C01815=1200.985,26.673,-44.909,-179.490,5.662,148.847
C01816=1200.990,26.424,-44.893,-179.493,5.662,148.848
C01817=1200.995,26.174,-44.879,-179.495,5.661,148.848
C01818=1201.000,25.924,-44.863,-179.498,5.660,148.849
C01819=1201.005,25.675,-44.848,-179.500,5.660,148.849
C01820=1201.009,25.425,-44.834,-179.503,5.659,148.850
C01821=1201.015,25.176,-44.818,-179.506,5.659,148.851
C01822=1201.019,24.926,-44.803,-179.508,5.658,148.851
C01823=1201.025,24.676,-44.788,-179.510,5.657,148.852
C01824=1201.030,24.427,-44.773,-179.513,5.657,148.853
C01825=1201.035,24.178,-44.758,-179.516,5.656,148.853
C01826=1201.040,23.928,-44.743,-179.518,5.656,148.854
C01827=1201.045,23.679,-44.728,-179.520,5.655,148.854
C01828=1201.050,23.430,-44.713,-179.523,5.654,148.855
C01829=1201.055,23.180,-44.698,-179.526,5.654,148.856
C01830=1201.060,22.931,-44.683,-179.528,5.653,148.856
C01831=1201.065,22.681,-44.669,-179.531,5.653,148.857
C01832=1201.070,22.432,-44.654,-179.533,5.652,148.858
C01833=1201.076,22.182,-44.639,-179.536,5.651,148.858
C01834=1201.080,21.932,-44.623,-179.539,5.651,148.859
C01835=1201.084,21.683,-44.608,-179.541,5.650,148.860
C01836=1201.090,21.433,-44.593,-179.544,5.650,148.860
C01837=1201.095,21.184,-44.578,-179.545,5.650,148.861
C01838=1201.100,20.934,-44.564,-179.548,5.649,148.861
C01839=1201.105,20.685,-44.549,-179.551,5.649,148.862
C01840=1201.110,20.435,-44.534,-179.553,5.648,148.863
C01841=1201.115,20.186,-44.519,-179.556,5.648,148.863
C01842=1201.120,19.936,-44.504,-179.558,5.647,148.864
C01843=1201.125,19.687,-44.489,-179.561,5.646,148.865
C01844=1201.130,19.437,-44.475,-179.563,5.646,148.865
C01845=1201.135,19.188,-44.460,-179.566,5.645,148.866
C01846=1201.140,18.938,-44.445,-179.569,5.645,148.867
C01847=1201.145,18.689,-44.430,-179.571,5.644,148.867
C01848=1201.150,18.439,-44.416,-179.574,5.644,148.868
C01849=1201.156,18.189,-44.401,-179.576,5.643,148.868
C01850=1201.160,17.940,-44.386,-179.579,5.643,148.869
C01851=1201.165,17.690,-44.372,-179.581,5.642,148.870
C01852=1201.170,17.441,-44.357,-179.584,5.641,148.870
C01853=1201.176,17.191,-44.342,-179.586,5.641,148.871
C01854=1201.180,16.942,-44.327,-179.589,5.640,148.872
C01855=1201.185,16.692,-44.313,-179.592,5.640,148.872
C01856=1201.191,16.443,-44.299,-179.594,5.639,148.873
C01857=1201.196,16.194,-44.283,-179.596,5.638,148.873
C01858=1201.201,15.944,-44.269,-179.599,5.638,148.874
C01859=1201.206,15.695,-44.255,-179.601,5.638,148.875
C01860=1201.211,15.446,-44.240,-179.604,5.638,148.876
C01861=1201.216,15.196,-44.225,-179.606,5.637,148.876
C01862=1201.221,14.946,-44.211,-179.609,5.636,148.877
C01863=1201.226,14.697,-44.196,-179.611,5.636,148.877
C01864=1201.231,14.447,-44.181,-179.614,5.635,148.878
C01865=1201.236,14.197,-44.167,-179.617,5.635,148.879
C01866=1201.240,13.948,-44.152,-179.619,5.634,148.879
C01867=1201.245,13.698,-44.138,-179.622,5.634,148.880
C01868=1201.251,13.448,-44.123,-179.624,5.633,148.881
C01869=1201.256,13.199,-44.109,-179.627,5.632,148.881
C01870=1201.261,12.950,-44.094,-179.629,5.632,148.882
C01871=1201.266,12.701,-44.080,-179.632,5.631,148.883
C01872=1201.271,12.451,-44.065,-179.635,5.631,148.883
C01873=1201.276,12.201,-44.051,-179.637,5.630,148.884
C01874=1201.281,11.952,-44.036,-179.639,5.630,148.884
C01875=1201.287,11.702,-44.021,-179.641,5.630,148.885
C01876=1201.291,11.452,-44.007,-179.644,5.629,148.886
C01877=1201.296,11.203,-43.993,-179.647,5.629,148.886
C01878=1201.301,10.954,-43.978,-179.649,5.628,148.887
C01879=1201.307,10.705,-43.964,-179.652,5.627,148.888
C01880=1201.312,10.455,-43.950,-179.654,5.627,148.888
C01881=1201.317,10.205,-43.935,-179.657,5.626,148.889
C01882=1201.322,9.955,-43.921,-179.660,5.626,148.890
C01883=1201.326,9.706,-43.907,-179.662,5.625,148.890
C01884=1201.331,9.457,-43.892,-179.664,5.624,148.891
C01885=1201.337,9.207,-43.877,-179.667,5.624,148.891
C01886=1201.342,8.958,-43.863,-179.669,5.624,148.892
C01887=1201.347,8.708,-43.849,-179.672,5.624,148.893
C01888=1201.352,8.458,-43.834,-179.674,5.623,148.894
C01889=1201.357,8.208,-43.820,-179.677,5.623,148.894
C01890=1201.362,7.959,-43.806,-179.679,5.622,148.895
C01891=1201.367,7.709,-43.792,-179.682,5.621,148.895
C01892=1201.373,7.460,-43.778,-179.684,5.621,148.896
C01893=1201.377,7.211,-43.763,-179.687,5.620,148.897
C01894=1201.382,6.961,-43.748,-179.690,5.620,148.897
C01895=1201.387,6.712,-43.734,-179.692,5.619,148.898
C01896=1201.392,6.462,-43.720,-179.694,5.619,148.899
C01897=1201.397,6.212,-43.706,-179.697,5.619,148.899
C01898=1201.403,5.963,-43.692,-179.699,5.618,148.900
C01899=1201.408,5.713,-43.677,-179.702,5.618,148.901
C01900=1201.413,5.464,-43.663,-179.705,5.617,148.901
C01901=1201.418,5.214,-43.649,-179.707,5.616,148.902
C01902=1201.423,4.964,-43.634,-179.709,5.616,148.902
C01903=1201.428,4.715,-43.621,-179.712,5.615,148.903
C01904=1201.433,4.466,-43.606,-179.715,5.615,148.904
C01905=1201.438,4.216,-43.592,-179.717,5.614,148.905
C01906=1201.442,3.966,-43.578,-179.719,5.615,148.905
C01907=1201.448,3.717,-43.564,-179.722,5.614,148.906
C01908=1201.453,3.468,-43.550,-179.724,5.613,148.906
C01909=1201.458,3.198,-43.535,-179.727,5.613,148.907
C01910=1201.464,2.929,-43.520,-179.730,5.612,148.908
C01911=1201.469,2.660,-43.504,-179.732,5.612,148.908
C01912=1201.475,2.391,-43.490,-179.735,5.611,148.909
C01913=1201.480,2.142,-43.476,-179.738,5.611,148.910
C01914=1201.485,1.892,-43.461,-179.740,5.610,148.910
C01915=1201.490,1.642,-43.447,-179.743,5.610,148.911
C01916=1201.495,1.393,-43.433,-179.746,5.609,148.912
C01917=1201.500,1.144,-43.419,-179.748,5.609,148.913
C01918=1201.505,0.893,-43.405,-179.750,5.608,148.913
C01919=1201.510,0.643,-43.391,-179.752,5.608,148.914
C01920=1201.516,0.394,-43.377,-179.755,5.608,148.914
C01921=1201.520,0.145,-43.363,-179.758,5.607,148.915
C01922=1201.525,-0.105,-43.349,-179.760,5.607,148.916
C01923=1201.531,-0.354,-43.335,-179.763,5.606,148.916
C01924=1201.536,-0.603,-43.321,-179.765,5.605,148.917
C01925=1201.541,-0.854,-43.307,-179.768,5.605,148.918
C01926=1201.546,-1.103,-43.293,-179.770,5.605,148.918
C01927=1201.551,-1.352,-43.280,-179.773,5.605,148.919
C01928=1201.556,-1.602,-43.265,-179.775,5.604,148.920
C01929=1201.561,-1.852,-43.251,-179.778,5.604,148.920
C01930=1201.566,-2.101,-43.238,-179.780,5.603,148.921
C01931=1201.571,-2.351,-43.224,-179.783,5.602,148.921
C01932=1201.576,-2.600,-43.210,-179.785,5.602,148.922
C01933=1201.581,-2.849,-43.196,-179.788,5.602,148.923
C01934=1201.586,-3.100,-43.183,-179.790,5.602,148.924
C01935=1201.591,-3.349,-43.168,-179.793,5.601,148.924
C01936=1201.597,-3.598,-43.154,-179.795,5.600,148.925
C01937=1201.601,-3.848,-43.141,-179.798,5.600,148.925
C01938=1201.606,-4.098,-43.127,-179.800,5.599,148.926
C01939=1201.612,-4.347,-43.113,-179.803,5.599,148.927
C01940=1201.617,-4.597,-43.099,-179.805,5.599,148.927
C01941=1201.622,-4.846,-43.086,-179.808,5.599,148.928
C01942=1201.627,-5.096,-43.072,-179.810,5.598,148.929
C01943=1201.632,-5.345,-43.058,-179.812,5.597,148.929
C01944=1201.638,-5.595,-43.045,-179.815,5.597,148.930
C01945=1201.642,-5.845,-43.031,-179.818,5.596,148.931
C01946=1201.647,-6.094,-43.017,-179.820,5.596,148.931
C01947=1201.653,-6.344,-43.003,-179.822,5.596,148.932
C01948=1201.657,-6.593,-42.990,-179.825,5.596,148.933
C01949=1201.663,-6.842,-42.976,-179.827,5.595,148.933
C01950=1201.668,-7.093,-42.962,-179.830,5.594,148.934
C01951=1201.672,-7.342,-42.949,-179.833,5.594,148.935
C01952=1201.678,-7.592,-42.935,-179.835,5.594,148.935
C01953=1201.683,-7.841,-42.921,-179.837,5.594,148.936
C01954=1201.688,-8.090,-42.908,-179.840,5.593,148.937
C01955=1201.693,-8.340,-42.894,-179.842,5.592,148.937
C01956=1201.698,-8.590,-42.880,-179.845,5.592,148.938
C01957=1201.703,-8.839,-42.867,-179.847,5.592,148.939
C01958=1201.708,-9.089,-42.853,-179.850,5.591,148.939
C01959=1201.714,-9.339,-42.840,-179.852,5.591,148.940
C01960=1201.718,-9.588,-42.826,-179.855,5.591,148.941
C01961=1201.724,-9.837,-42.812,-179.857,5.590,148.941
C01962=1201.729,-10.087,-42.799,-179.860,5.590,148.942
C01963=1201.733,-10.337,-42.785,-179.862,5.589,148.942
C01964=1201.739,-10.586,-42.772,-179.865,5.589,148.943
C01965=1201.743,-10.836,-42.758,-179.867,5.589,148.944
C01966=1201.749,-11.086,-42.745,-179.870,5.588,148.945
C01967=1201.754,-11.335,-42.731,-179.872,5.588,148.945
C01968=1201.759,-11.585,-42.718,-179.875,5.587,148.946
C01969=1201.764,-11.834,-42.704,-179.877,5.587,148.946
C01970=1201.769,-12.084,-42.691,-179.879,5.587,148.947
C01971=1201.774,-12.334,-42.678,-179.882,5.586,148.948
C01972=1201.779,-12.583,-42.664,-179.885,5.586,148.948
C01973=1201.785,-12.833,-42.651,-179.887,5.585,148.949
C01974=1201.790,-13.082,-42.637,-179.890,5.585,148.950
C01975=1201.795,-13.332,-42.624,-179.891,5.585,148.950
C01976=1201.800,-13.582,-42.610,-179.894,5.584,148.951
C01977=1201.805,-13.831,-42.597,-179.897,5.584,148.952
C01978=1201.810,-14.081,-42.583,-179.899,5.583,148.952
C01979=1201.815,-14.330,-42.570,-179.902,5.583,148.953
C01980=1201.820,-14.580,-42.557,-179.905,5.582,148.954
C01981=1201.825,-14.829,-42.543,-179.906,5.582,148.954
C01982=1201.831,-15.079,-42.530,-179.909,5.582,148.955
C01983=1201.835,-15.329,-42.517,-179.912,5.581,148.956
C01984=1201.841,-15.578,-42.503,-179.914,5.581,148.956
C01985=1201.845,-15.828,-42.490,-179.917,5.581,148.957
C01986=1201.851,-16.077,-42.477,-179.919,5.581,148.958
C01987=1201.855,-16.327,-42.463,-179.922,5.580,148.958
C01988=1201.861,-16.576,-42.450,-179.924,5.580,148.959
C01989=1201.866,-16.826,-42.437,-179.927,5.579,148.960
C01990=1201.871,-17.075,-42.423,-179.929,5.579,148.960
C01991=1201.876,-17.325,-42.410,-179.931,5.579,148.961
C01992=1201.882,-17.575,-42.397,-179.934,5.578,148.962
C01993=1201.886,-17.825,-42.384,-179.937,5.578,148.962
C01994=1201.892,-18.074,-42.370,-179.939,5.577,148.963
C01995=1201.897,-18.323,-42.358,-179.941,5.577,148.963
C01996=1201.902,-18.574,-42.344,-179.943,5.577,148.964
C01997=1201.907,-18.823,-42.331,-179.946,5.576,148.965
C01998=1201.912,-19.072,-42.318,-179.949,5.576,148.966
C01999=1201.917,-19.322,-42.305,-179.951,5.575,148.966
C02000=1201.922,-19.572,-42.292,-179.954,5.576,148.967
C02001=1201.928,-19.822,-42.278,-179.956,5.575,148.967
C02002=1201.933,-20.070,-42.265,-179.958,5.574,148.968
C02003=1201.937,-20.320,-42.252,-179.961,5.574,148.969
C02004=1201.943,-20.570,-42.239,-179.964,5.574,148.970
C02005=1201.947,-20.820,-42.226,-179.966,5.574,148.970
C02006=1201.953,-21.070,-42.213,-179.968,5.573,148.971
C02007=1201.958,-21.318,-42.200,-179.971,5.573,148.972
C02008=1201.963,-21.568,-42.187,-179.973,5.572,148.972
C02009=1201.969,-21.818,-42.173,-179.975,5.572,148.973
C02010=1201.973,-22.068,-42.160,-179.978,5.572,148.973
C02011=1201.978,-22.317,-42.148,-179.981,5.571,148.974
C02012=1201.984,-22.567,-42.135,-179.983,5.571,148.975
C02013=1201.989,-22.836,-42.120,-179.986,5.570,148.976
C02014=1201.994,-23.106,-42.106,-179.989,5.570,148.976
C02015=1202.000,-23.375,-42.093,-179.991,5.570,148.977
C02016=1202.006,-23.645,-42.078,-179.993,5.570,148.978
C02017=1202.011,-23.895,-42.066,-179.996,5.569,148.978
C02018=1202.016,-24.145,-42.052,-179.999,5.569,148.979
C02019=1202.021,-24.394,-42.040,179.999,5.568,148.980
C02020=1202.026,-24.644,-42.026,179.997,5.569,148.980
C02021=1202.031,-24.893,-42.013,179.994,5.568,148.981
C02022=1202.037,-25.143,-42.000,179.992,5.567,148.982
C02023=1202.041,-25.393,-41.987,179.989,5.567,148.982
C02024=1202.046,-25.642,-41.975,179.986,5.567,148.983
C02025=1202.052,-25.892,-41.961,179.984,5.567,148.984
C02026=1202.057,-26.142,-41.948,179.982,5.566,148.984
C02027=1202.062,-26.391,-41.936,179.979,5.566,148.985
C02028=1202.067,-26.640,-41.923,179.977,5.565,148.986
C02029=1202.072,-26.891,-41.910,179.975,5.565,148.986
C02030=1202.077,-27.140,-41.897,179.972,5.565,148.987
C02031=1202.082,-27.389,-41.884,179.969,5.564,148.988
C02032=1202.087,-27.638,-41.872,179.967,5.564,148.988
C02033=1202.093,-27.889,-41.858,179.965,5.564,148.989
C02034=1202.098,-28.138,-41.846,179.963,5.563,148.989
C02035=1202.103,-28.387,-41.833,179.960,5.563,148.990
C02036=1202.107,-28.637,-41.820,179.957,5.563,148.991
C02037=1202.113,-28.887,-41.807,179.955,5.563,148.992
C02038=1202.118,-29.136,-41.794,179.952,5.562,148.992
C02039=1202.124,-29.386,-41.782,179.950,5.562,148.993
C02040=1202.128,-29.636,-41.769,179.947,5.561,148.994
C02041=1202.134,-29.886,-41.757,179.946,5.561,148.994
C02042=1202.139,-30.135,-41.744,179.943,5.561,148.995
C02043=1202.144,-30.385,-41.731,179.940,5.560,148.996
C02044=1202.149,-30.635,-41.718,179.938,5.560,148.996
C02045=1202.154,-30.884,-41.705,179.935,5.560,148.997
C02046=1202.159,-31.133,-41.693,179.933,5.560,148.998
C02047=1202.164,-31.383,-41.680,179.930,5.559,148.998
C02048=1202.169,-31.633,-41.667,179.929,5.559,148.999
C02049=1202.175,-31.883,-41.655,179.926,5.559,148.999
C02050=1202.180,-32.132,-41.642,179.923,5.558,149.000
C02051=1202.185,-32.382,-41.629,179.921,5.558,149.001
C02052=1202.190,-32.631,-41.617,179.919,5.558,149.002
C02053=1202.195,-32.881,-41.604,179.916,5.558,149.002
C02054=1202.200,-33.131,-41.592,179.913,5.557,149.003
C02055=1202.206,-33.380,-41.580,179.911,5.557,149.003
C02056=1202.211,-33.630,-41.566,179.909,5.557,149.004
C02057=1202.216,-33.880,-41.553,179.906,5.556,149.005
C02058=1202.221,-34.129,-41.541,179.904,5.556,149.006
C02059=1202.227,-34.379,-41.529,179.902,5.556,149.006
C02060=1202.232,-34.628,-41.516,179.899,5.556,149.007
C02061=1202.236,-34.878,-41.503,179.896,5.555,149.008
C02062=1202.241,-35.128,-41.491,179.894,5.555,149.008
C02063=1202.247,-35.378,-41.479,179.892,5.555,149.009
C02064=1202.252,-35.627,-41.466,179.889,5.554,149.010
C02065=1202.257,-35.876,-41.454,179.887,5.554,149.010
C02066=1202.261,-36.126,-41.441,179.884,5.553,149.011
C02067=1202.267,-36.376,-41.429,179.882,5.554,149.012
C02068=1202.272,-36.625,-41.416,179.880,5.553,149.012
C02069=1202.278,-36.875,-41.403,179.877,5.552,149.013
C02070=1202.283,-37.125,-41.391,179.875,5.553,149.013
C02071=1202.288,-37.374,-41.378,179.872,5.552,149.014
C02072=1202.293,-37.624,-41.366,179.870,5.552,149.015
C02073=1202.298,-37.874,-41.353,179.867,5.551,149.016
C02074=1202.304,-38.124,-41.341,179.865,5.552,149.016
C02075=1202.309,-38.373,-41.328,179.863,5.551,149.017
C02076=1202.314,-38.623,-41.317,179.860,5.550,149.017
C02077=1202.319,-38.872,-41.304,179.858,5.551,149.018
C02078=1202.324,-39.121,-41.291,179.855,5.550,149.019
C02079=1202.329,-39.372,-41.279,179.853,5.550,149.020
C02080=1202.334,-39.621,-41.267,179.850,5.549,149.020
C02081=1202.339,-39.871,-41.254,179.848,5.550,149.021
C02082=1202.345,-40.121,-41.242,179.846,5.549,149.021
C02083=1202.350,-40.370,-41.229,179.843,5.548,149.022
C02084=1202.355,-40.620,-41.218,179.841,5.549,149.023
C02085=1202.360,-40.869,-41.206,179.838,5.548,149.024
C02086=1202.365,-41.118,-41.193,179.836,5.548,149.024
C02087=1202.370,-41.369,-41.181,179.834,5.548,149.025
C02088=1202.375,-41.618,-41.168,179.831,5.547,149.025
C02089=1202.380,-41.868,-41.156,179.829,5.547,149.026
C02090=1202.385,-42.117,-41.144,179.826,5.547,149.027
C02091=1202.391,-42.367,-41.132,179.824,5.547,149.028
C02092=1202.396,-42.617,-41.119,179.821,5.546,149.028
C02093=1202.401,-42.867,-41.107,179.819,5.546,149.029
C02094=1202.407,-43.116,-41.095,179.817,5.546,149.030
C02095=1202.412,-43.366,-41.083,179.814,5.545,149.030
C02096=1202.417,-43.615,-41.070,179.812,5.545,149.031
C02097=1202.422,-43.865,-41.059,179.810,5.545,149.031
C02098=1202.426,-44.115,-41.046,179.807,5.545,149.032
C02099=1202.432,-44.365,-41.034,179.804,5.544,149.033
C02100=1202.437,-44.614,-41.021,179.802,5.545,149.034
C02101=1202.442,-44.864,-41.010,179.800,5.544,149.034
C02102=1202.447,-45.113,-40.997,179.797,5.543,149.035
C02103=1202.453,-45.363,-40.985,179.795,5.543,149.035
C02104=1202.458,-45.613,-40.972,179.793,5.543,149.036
C02105=1202.463,-45.862,-40.961,179.790,5.543,149.037
C02106=1202.468,-46.112,-40.949,179.787,5.542,149.038
C02107=1202.473,-46.362,-40.937,179.785,5.543,149.038
C02108=1202.479,-46.611,-40.925,179.783,5.542,149.039
C02109=1202.484,-46.861,-40.912,179.780,5.542,149.039
C02110=1202.489,-47.111,-40.900,179.778,5.542,149.040
C02111=1202.494,-47.360,-40.889,179.776,5.541,149.041
C02112=1202.499,-47.610,-40.876,179.773,5.541,149.042
C02113=1202.504,-47.860,-40.864,179.771,5.541,149.042
C02114=1202.510,-48.109,-40.852,179.769,5.540,149.043
C02115=1202.515,-48.359,-40.840,179.766,5.540,149.043
C02116=1202.520,-48.608,-40.829,179.764,5.540,149.044
C02117=1202.526,-48.879,-40.815,179.761,5.540,149.045
C02118=1202.532,-49.149,-40.803,179.759,5.539,149.046
C02119=1202.537,-49.419,-40.789,179.756,5.539,149.046
C02120=1202.542,-49.689,-40.776,179.753,5.539,149.047
C02121=1202.547,-49.939,-40.764,179.751,5.539,149.048
C02122=1202.552,-50.188,-40.753,179.749,5.538,149.048
C02123=1202.557,-50.438,-40.740,179.746,5.538,149.049
C02124=1202.563,-50.688,-40.728,179.744,5.538,149.050
C02125=1202.568,-50.938,-40.716,179.741,5.538,149.050
C02126=1202.573,-51.187,-40.705,179.739,5.537,149.051
C02127=1202.578,-51.437,-40.692,179.737,5.537,149.052
C02128=1202.584,-51.686,-40.681,179.734,5.537,149.052
C02129=1202.589,-51.936,-40.669,179.732,5.537,149.053
C02130=1202.594,-52.185,-40.658,179.730,5.537,149.054
C02131=1202.599,-52.435,-40.645,179.727,5.536,149.054
C02132=1202.605,-52.685,-40.633,179.724,5.536,149.055
C02133=1202.609,-52.934,-40.622,179.723,5.536,149.056
C02134=1202.615,-53.184,-40.610,179.720,5.535,149.056
C02135=1202.620,-53.434,-40.598,179.717,5.535,149.057
C02136=1202.624,-53.683,-40.586,179.715,5.535,149.058
C02137=1202.630,-53.933,-40.574,179.712,5.535,149.058
C02138=1202.635,-54.183,-40.562,179.710,5.535,149.059
C02139=1202.640,-54.433,-40.551,179.708,5.534,149.060
C02140=1202.645,-54.682,-40.539,179.706,5.534,149.060
C02141=1202.651,-54.932,-40.527,179.703,5.534,149.061
C02142=1202.655,-55.182,-40.515,179.701,5.534,149.062
C02143=1202.661,-55.431,-40.504,179.698,5.533,149.062
C02144=1202.666,-55.681,-40.492,179.696,5.534,149.063
C02145=1202.671,-55.930,-40.481,179.694,5.533,149.064
C02146=1202.677,-56.180,-40.469,179.691,5.533,149.064
C02147=1202.682,-56.430,-40.456,179.689,5.533,149.065
C02148=1202.687,-56.679,-40.445,179.686,5.532,149.066
C02149=1202.692,-56.929,-40.433,179.684,5.532,149.066
C02150=1202.697,-57.179,-40.422,179.682,5.532,149.067
C02151=1202.702,-57.429,-40.410,179.680,5.532,149.068
C02152=1202.708,-57.679,-40.398,179.677,5.531,149.068
C02153=1202.712,-57.928,-40.387,179.675,5.531,149.069
C02154=1202.718,-58.178,-40.375,179.672,5.531,149.070
C02155=1202.723,-58.427,-40.364,179.670,5.531,149.070
C02156=1202.728,-58.677,-40.352,179.667,5.531,149.071
C02157=1202.733,-58.927,-40.341,179.665,5.530,149.072
C02158=1202.738,-59.176,-40.328,179.663,5.530,149.072
C02159=1202.744,-59.426,-40.316,179.660,5.530,149.073
C02160=1202.748,-59.676,-40.305,179.658,5.530,149.074
C02161=1202.754,-59.925,-40.293,179.656,5.530,149.074
C02162=1202.759,-60.174,-40.282,179.653,5.529,149.075
C02163=1202.765,-60.424,-40.270,179.651,5.529,149.076
C02164=1202.769,-60.674,-40.259,179.649,5.529,149.076
C02165=1202.775,-60.924,-40.247,179.646,5.529,149.077
C02166=1202.779,-61.174,-40.236,179.644,5.529,149.078
C02167=1202.785,-61.423,-40.224,179.641,5.528,149.078
C02168=1202.790,-61.672,-40.213,179.639,5.528,149.079
C02169=1202.796,-61.922,-40.201,179.637,5.528,149.080
C02170=1202.801,-62.173,-40.190,179.634,5.528,149.080
C02171=1202.806,-62.423,-40.179,179.632,5.527,149.081
C02172=1202.811,-62.672,-40.167,179.630,5.527,149.082
C02173=1202.817,-62.921,-40.156,179.627,5.527,149.082
C02174=1202.821,-63.171,-40.145,179.625,5.527,149.083
C02175=1202.827,-63.421,-40.133,179.623,5.527,149.084
C02176=1202.832,-63.671,-40.121,179.620,5.526,149.084
C02177=1202.837,-63.921,-40.109,179.618,5.526,149.085
C02178=1202.842,-64.169,-40.099,179.615,5.526,149.086
C02179=1202.848,-64.419,-40.087,179.613,5.526,149.086
C02180=1202.852,-64.669,-40.075,179.611,5.526,149.087
C02181=1202.858,-64.919,-40.063,179.608,5.525,149.088
C02182=1202.863,-65.169,-40.053,179.606,5.526,149.088
C02183=1202.869,-65.418,-40.041,179.604,5.525,149.089
C02184=1202.874,-65.668,-40.030,179.601,5.525,149.090
C02185=1202.878,-65.918,-40.019,179.599,5.525,149.090
C02186=1202.884,-66.168,-40.007,179.597,5.524,149.091
C02187=1202.889,-66.417,-39.996,179.594,5.524,149.092
C02188=1202.894,-66.666,-39.984,179.592,5.524,149.092
C02189=1202.899,-66.917,-39.974,179.589,5.524,149.093
C02190=1202.904,-67.166,-39.962,179.587,5.524,149.094
C02191=1202.910,-67.416,-39.951,179.585,5.524,149.094
C02192=1202.915,-67.665,-39.939,179.582,5.523,149.095
C02193=1202.920,-67.915,-39.928,179.580,5.523,149.096
C02194=1202.925,-68.165,-39.917,179.578,5.523,149.096
C02195=1202.930,-68.414,-39.906,179.576,5.523,149.097
C02196=1202.936,-68.664,-39.894,179.573,5.523,149.098
C02197=1202.941,-68.914,-39.883,179.571,5.522,149.098
C02198=1202.947,-69.164,-39.872,179.569,5.522,149.099
C02199=1202.952,-69.413,-39.861,179.566,5.522,149.100
C02200=1202.956,-69.663,-39.849,179.564,5.522,149.100
C02201=1202.962,-69.913,-39.838,179.561,5.522,149.101
C02202=1202.967,-70.162,-39.827,179.559,5.521,149.102
C02203=1202.972,-70.412,-39.816,179.557,5.521,149.102
C02204=1202.977,-70.662,-39.804,179.554,5.521,149.103
C02205=1202.983,-70.911,-39.793,179.552,5.521,149.104
C02206=1202.988,-71.161,-39.783,179.549,5.521,149.104
C02207=1202.993,-71.411,-39.771,179.547,5.520,149.105
C02208=1202.998,-71.660,-39.760,179.545,5.520,149.106
C02209=1203.003,-71.910,-39.749,179.543,5.520,149.106
C02210=1203.009,-72.160,-39.737,179.540,5.520,149.107
C02211=1203.014,-72.409,-39.727,179.538,5.520,149.108
C02212=1203.019,-72.659,-39.716,179.535,5.519,149.108
C02213=1203.024,-72.909,-39.705,179.533,5.519,149.109
C02214=1203.030,-73.158,-39.693,179.531,5.519,149.110
C02215=1203.035,-73.409,-39.683,179.529,5.519,149.110
C02216=1203.040,-73.658,-39.671,179.526,5.519,149.111
C02217=1203.046,-73.908,-39.660,179.523,5.518,149.112
C02218=1203.051,-74.158,-39.649,179.522,5.518,149.112
C02219=1203.055,-74.407,-39.638,179.519,5.518,149.113
C02220=1203.061,-74.657,-39.628,179.517,5.518,149.114
C02221=1203.067,-74.928,-39.615,179.514,5.518,149.114
C02222=1203.072,-75.199,-39.603,179.512,5.517,149.115
C02223=1203.078,-75.469,-39.591,179.510,5.518,149.116
C02224=1203.083,-75.740,-39.580,179.507,5.517,149.116
C02225=1203.089,-75.990,-39.568,179.504,5.517,149.117
C02226=1203.094,-76.239,-39.558,179.502,5.517,149.118
C02227=1203.099,-76.489,-39.546,179.500,5.517,149.119
C02228=1203.105,-76.738,-39.536,179.497,5.516,149.119
C02229=1203.110,-76.988,-39.524,179.495,5.516,149.120
C02230=1203.115,-77.239,-39.514,179.493,5.516,149.120
C02231=1203.120,-77.487,-39.503,179.490,5.516,149.121
C02232=1203.125,-77.738,-39.492,179.488,5.516,149.122
C02233=1203.131,-77.987,-39.481,179.486,5.516,149.122
C02234=1203.136,-78.237,-39.470,179.484,5.515,149.123
C02235=1203.141,-78.487,-39.459,179.481,5.515,149.124
C02236=1203.147,-78.736,-39.448,179.479,5.515,149.124
C02237=1203.151,-78.986,-39.437,179.476,5.515,149.125
C02238=1203.157,-79.236,-39.427,179.475,5.515,149.126
C02239=1203.162,-79.485,-39.416,179.472,5.515,149.126
C02240=1203.168,-79.735,-39.405,179.470,5.515,149.127
C02241=1203.173,-79.985,-39.394,179.467,5.514,149.128
C02242=1203.178,-80.235,-39.383,179.465,5.514,149.128
C02243=1203.183,-80.484,-39.372,179.463,5.514,149.129
C02244=1203.188,-80.734,-39.362,179.460,5.514,149.130
C02245=1203.194,-80.984,-39.351,179.458,5.514,149.130
C02246=1203.198,-81.233,-39.340,179.455,5.514,149.131
C02247=1203.204,-81.483,-39.330,179.454,5.514,149.132
C02248=1203.209,-81.733,-39.318,179.451,5.513,149.132
C02249=1203.214,-81.983,-39.307,179.448,5.513,149.133
C02250=1203.220,-82.232,-39.297,179.446,5.513,149.134
C02251=1203.225,-82.482,-39.286,179.444,5.513,149.134
C02252=1203.230,-82.732,-39.276,179.442,5.513,149.135
C02253=1203.235,-82.981,-39.264,179.439,5.512,149.136
C02254=1203.240,-83.231,-39.254,179.437,5.513,149.136
C02255=1203.245,-83.481,-39.244,179.435,5.512,149.137
C02256=1203.251,-83.730,-39.233,179.432,5.512,149.138
C02257=1203.256,-83.980,-39.222,179.430,5.512,149.138
C02258=1203.261,-84.230,-39.212,179.428,5.511,149.139
C02259=1203.266,-84.479,-39.201,179.426,5.512,149.140
C02260=1203.272,-84.729,-39.190,179.423,5.511,149.140
C02261=1203.277,-84.979,-39.180,179.421,5.511,149.141
C02262=1203.283,-85.228,-39.168,179.419,5.511,149.142
C02263=1203.288,-85.479,-39.158,179.417,5.511,149.142
C02264=1203.293,-85.728,-39.148,179.414,5.511,149.143
C02265=1203.298,-85.978,-39.137,179.411,5.510,149.144
C02266=1203.303,-86.227,-39.126,179.410,5.510,149.144
C02267=1203.308,-86.478,-39.115,179.407,5.510,149.145
C02268=1203.314,-86.727,-39.105,179.405,5.510,149.146
C02269=1203.319,-86.977,-39.094,179.402,5.510,149.146
C02270=1203.324,-87.226,-39.084,179.401,5.510,149.147
C02271=1203.329,-87.477,-39.073,179.398,5.509,149.148
C02272=1203.335,-87.726,-39.063,179.396,5.510,149.148
C02273=1203.340,-87.976,-39.052,179.393,5.509,149.149
C02274=1203.345,-88.225,-39.041,179.391,5.509,149.149
C02275=1203.350,-88.476,-39.031,179.389,5.509,149.150
C02276=1203.356,-88.725,-39.021,179.386,5.508,149.151
C02277=1203.360,-88.975,-39.011,179.384,5.509,149.152
C02278=1203.365,-89.224,-39.000,179.381,5.508,149.152
C02279=1203.371,-89.473,-38.990,179.380,5.508,149.153
C02280=1203.376,-89.724,-38.979,179.377,5.508,149.153
C02281=1203.382,-89.973,-38.969,179.375,5.508,149.154
C02282=1203.387,-90.224,-38.958,179.372,5.508,149.155
C02283=1203.392,-90.472,-38.947,179.371,5.508,149.155
C02284=1203.397,-90.723,-38.937,179.368,5.508,149.156
C02285=1203.402,-90.972,-38.926,179.366,5.507,149.157
C02286=1203.407,-91.222,-38.916,179.363,5.507,149.157
C02287=1203.413,-91.472,-38.906,179.361,5.507,149.158
C02288=1203.419,-91.722,-38.895,179.359,5.507,149.159
C02289=1203.424,-91.972,-38.885,179.356,5.507,149.159
C02290=1203.429,-92.221,-38.875,179.354,5.507,149.160
C02291=1203.433,-92.471,-38.864,179.352,5.506,149.161
C02292=1203.439,-92.720,-38.854,179.350,5.507,149.161
C02293=1203.444,-92.970,-38.844,179.347,5.506,149.162
C02294=1203.449,-93.220,-38.833,179.345,5.507,149.163
C02295=1203.455,-93.470,-38.823,179.343,5.506,149.163
C02296=1203.460,-93.720,-38.812,179.341,5.506,149.164
C02297=1203.466,-93.969,-38.802,179.338,5.506,149.165
C02298=1203.471,-94.219,-38.792,179.336,5.506,149.165
C02299=1203.476,-94.469,-38.781,179.334,5.505,149.166
C02300=1203.481,-94.718,-38.772,179.331,5.505,149.167
C02301=1203.487,-94.968,-38.761,179.329,5.505,149.167
C02302=1203.492,-95.218,-38.751,179.327,5.505,149.168
C02303=1203.497,-95.468,-38.741,179.325,5.505,149.168
C02304=1203.502,-95.718,-38.730,179.322,5.504,149.169
C02305=1203.508,-95.967,-38.720,179.320,5.505,149.170
C02306=1203.513,-96.217,-38.710,179.318,5.504,149.171
C02307=1203.518,-96.467,-38.700,179.316,5.504,149.171
C02308=1203.523,-96.716,-38.689,179.313,5.504,149.172
C02309=1203.529,-96.966,-38.679,179.311,5.504,149.172
C02310=1203.534,-97.216,-38.669,179.309,5.504,149.173
C02311=1203.539,-97.465,-38.659,179.307,5.504,149.174
C02312=1203.544,-97.715,-38.649,179.304,5.504,149.174
C02313=1203.549,-97.965,-38.638,179.302,5.504,149.175
C02314=1203.555,-98.215,-38.628,179.300,5.503,149.176
C02315=1203.561,-98.464,-38.618,179.298,5.503,149.176
C02316=1203.565,-98.714,-38.608,179.295,5.503,149.177
C02317=1203.570,-98.964,-38.598,179.293,5.503,149.178
C02318=1203.576,-99.213,-38.587,179.291,5.503,149.178
C02319=1203.581,-99.464,-38.577,179.288,5.502,149.179
C02320=1203.586,-99.713,-38.567,179.286,5.503,149.180
C02321=1203.591,-99.962,-38.557,179.284,5.502,149.180
C02322=1203.596,-100.213,-38.546,179.282,5.503,149.181
C02323=1203.602,-100.463,-38.537,179.279,5.502,149.182
C02324=1203.607,-100.712,-38.527,179.277,5.502,149.182
C02325=1203.613,-100.984,-38.516,179.275,5.502,149.183
C02326=1203.618,-101.255,-38.505,179.272,5.502,149.184
C02327=1203.625,-101.526,-38.494,179.270,5.502,149.184
C02328=1203.630,-101.797,-38.483,179.267,5.501,149.185
C02329=1203.636,-102.047,-38.473,179.265,5.502,149.186
C02330=1203.640,-102.297,-38.463,179.263,5.501,149.186
C02331=1203.646,-102.547,-38.453,179.261,5.501,149.187
C02332=1203.651,-102.796,-38.443,179.258,5.501,149.188
C02333=1203.656,-103.046,-38.433,179.256,5.501,149.188
C02334=1203.661,-103.296,-38.423,179.254,5.500,149.189
C02335=1203.667,-103.546,-38.413,179.252,5.501,149.190
C02336=1203.673,-103.796,-38.403,179.249,5.500,149.190
C02337=1203.678,-104.045,-38.393,179.247,5.500,149.191
C02338=1203.683,-104.295,-38.383,179.245,5.500,149.192
C02339=1203.688,-104.544,-38.373,179.243,5.500,149.192
C02340=1203.693,-104.794,-38.364,179.240,5.500,149.193
C02341=1203.699,-105.044,-38.354,179.238,5.500,149.193
C02342=1203.703,-105.294,-38.344,179.236,5.500,149.194
C02343=1203.709,-105.543,-38.333,179.234,5.500,149.195
C02344=1203.715,-105.794,-38.324,179.231,5.499,149.195
C02345=1203.720,-106.043,-38.314,179.229,5.500,149.196
C02346=1203.725,-106.293,-38.304,179.227,5.499,149.197
C02347=1203.730,-106.543,-38.293,179.225,5.500,149.198
C02348=1203.735,-106.792,-38.285,179.222,5.499,149.198
C02349=1203.741,-107.042,-38.274,179.220,5.499,149.199
C02350=1203.745,-107.292,-38.264,179.218,5.499,149.199
C02351=1203.751,-107.542,-38.255,179.216,5.499,149.200
C02352=1203.757,-107.792,-38.245,179.213,5.498,149.201
C02353=1203.762,-108.041,-38.235,179.211,5.499,149.201
C02354=1203.768,-108.291,-38.226,179.209,5.498,149.202
C02355=1203.772,-108.541,-38.216,179.207,5.498,149.203
C02356=1203.777,-108.790,-38.205,179.204,5.498,149.203
C02357=1203.783,-109.040,-38.195,179.202,5.498,149.204
C02358=1203.788,-109.290,-38.186,179.200,5.497,149.204
C02359=1203.794,-109.539,-38.176,179.198,5.498,149.205
C02360=1203.799,-109.789,-38.167,179.195,5.497,149.206
C02361=1203.804,-110.040,-38.157,179.194,5.497,149.206
C02362=1203.809,-110.289,-38.147,179.191,5.497,149.207
C02363=1203.815,-110.539,-38.137,179.189,5.497,149.208
C02364=1203.820,-110.788,-38.128,179.187,5.497,149.208
C02365=1203.825,-111.038,-38.118,179.185,5.497,149.209
C02366=1203.831,-111.288,-38.108,179.182,5.497,149.210
C02367=1203.835,-111.538,-38.098,179.180,5.497,149.210
C02368=1203.841,-111.788,-38.089,179.178,5.496,149.211
C02369=1203.846,-112.037,-38.079,179.176,5.497,149.212
C02370=1203.852,-112.287,-38.069,179.173,5.496,149.212
C02371=1203.857,-112.537,-38.060,179.171,5.496,149.213
C02372=1203.862,-112.786,-38.050,179.169,5.496,149.214
C02373=1203.868,-113.036,-38.041,179.167,5.496,149.214
C02374=1203.873,-113.286,-38.030,179.164,5.495,149.215
C02375=1203.878,-113.536,-38.021,179.162,5.496,149.215
C02376=1203.883,-113.786,-38.011,179.160,5.495,149.216
C02377=1203.889,-114.035,-38.002,179.158,5.495,149.217
C02378=1203.894,-114.285,-37.992,179.155,5.495,149.217
C02379=1203.899,-114.535,-37.983,179.153,5.495,149.218
C02380=1203.905,-114.784,-37.973,179.151,5.495,149.219
C02381=1203.910,-115.034,-37.964,179.149,5.495,149.219
C02382=1203.914,-115.284,-37.954,179.146,5.495,149.220
C02383=1203.920,-115.534,-37.945,179.145,5.495,149.220
C02384=1203.925,-115.784,-37.935,179.142,5.494,149.221
C02385=1203.931,-116.034,-37.925,179.140,5.495,149.222
C02386=1203.936,-116.283,-37.916,179.138,5.494,149.222
C02387=1203.942,-116.533,-37.906,179.136,5.494,149.223
C02388=1203.947,-116.782,-37.897,179.134,5.495,149.224
C02389=1203.953,-117.033,-37.887,179.131,5.494,149.224
C02390=1203.957,-117.282,-37.878,179.129,5.494,149.225
C02391=1203.963,-117.532,-37.869,179.127,5.494,149.226
C02392=1203.968,-117.781,-37.859,179.125,5.494,149.226
C02393=1203.973,-118.032,-37.849,179.122,5.493,149.227
C02394=1203.979,-118.282,-37.840,179.120,5.494,149.228
C02395=1203.983,-118.531,-37.830,179.118,5.493,149.228
C02396=1203.989,-118.781,-37.821,179.116,5.493,149.229
C02397=1203.994,-119.031,-37.811,179.113,5.493,149.230
C02398=1203.999,-119.280,-37.802,179.112,5.493,149.230
C02399=1204.005,-119.530,-37.793,179.109,5.493,149.231
C02400=1204.010,-119.780,-37.783,179.107,5.493,149.232
C02401=1204.015,-120.030,-37.774,179.105,5.492,149.232
C02402=1204.021,-120.279,-37.764,179.103,5.493,149.233
C02403=1204.026,-120.529,-37.755,179.100,5.492,149.233
C02404=1204.031,-120.779,-37.746,179.098,5.492,149.234
C02405=1204.037,-121.028,-37.736,179.096,5.492,149.235
C02406=1204.042,-121.278,-37.727,179.094,5.492,149.235
C02407=1204.047,-121.528,-37.718,179.092,5.492,149.236
C02408=1204.053,-121.778,-37.708,179.089,5.492,149.237
C02409=1204.058,-122.027,-37.699,179.087,5.492,149.237
C02410=1204.063,-122.277,-37.690,179.085,5.491,149.238
C02411=1204.069,-122.527,-37.680,179.083,5.492,149.238
C02412=1204.074,-122.777,-37.671,179.080,5.491,149.239
C02413=1204.079,-123.027,-37.662,179.079,5.491,149.240
C02414=1204.085,-123.277,-37.653,179.076,5.491,149.240
C02415=1204.090,-123.526,-37.643,179.074,5.491,149.241
C02416=1204.095,-123.776,-37.634,179.072,5.491,149.242
C02417=1204.100,-124.026,-37.625,179.070,5.491,149.242
C02418=1204.106,-124.275,-37.615,179.067,5.490,149.243
C02419=1204.111,-124.525,-37.606,179.065,5.491,149.244
C02420=1204.116,-124.775,-37.597,179.063,5.490,149.244
C02421=1204.122,-125.025,-37.588,179.061,5.490,149.245
C02422=1204.127,-125.274,-37.578,179.059,5.491,149.245
C02423=1204.132,-125.524,-37.569,179.056,5.490,149.246
C02424=1204.137,-125.774,-37.560,179.055,5.490,149.247
C02425=1204.143,-126.024,-37.551,179.052,5.490,149.247
C02426=1204.148,-126.274,-37.542,179.050,5.490,149.248
C02427=1204.153,-126.523,-37.532,179.048,5.490,149.249
C02428=1204.158,-126.773,-37.523,179.046,5.490,149.249
C02429=1203.738,-126.784,-37.562,179.042,5.493,149.251
C02430=1203.732,-126.534,-37.571,179.044,5.493,149.250
C02431=1203.727,-126.284,-37.580,179.046,5.494,149.250
C02432=1203.721,-126.035,-37.589,179.048,5.493,149.249
C02433=1203.716,-125.785,-37.597,179.050,5.494,149.249
C02434=1203.710,-125.536,-37.608,179.052,5.494,149.248
C02435=1203.705,-125.286,-37.617,179.055,5.494,149.247
C02436=1203.700,-125.036,-37.625,179.057,5.494,149.247
C02437=1203.695,-124.786,-37.634,179.059,5.493,149.246
C02438=1203.689,-124.537,-37.645,179.061,5.494,149.245
C02439=1203.684,-124.287,-37.653,179.063,5.494,149.245
C02440=1203.679,-124.037,-37.662,179.066,5.494,149.244
C02441=1203.673,-123.787,-37.672,179.068,5.494,149.243
C02442=1203.668,-123.538,-37.681,179.070,5.495,149.243
C02443=1203.663,-123.288,-37.690,179.072,5.494,149.242
C02444=1203.658,-123.038,-37.699,179.074,5.495,149.242
C02445=1203.652,-122.788,-37.709,179.076,5.495,149.241
C02446=1203.647,-122.539,-37.718,179.079,5.495,149.240
C02447=1203.642,-122.289,-37.727,179.081,5.495,149.240
C02448=1203.636,-122.039,-37.737,179.083,5.495,149.239
C02449=1203.631,-121.789,-37.746,179.085,5.495,149.238
C02450=1203.626,-121.539,-37.755,179.088,5.496,149.238
C02451=1203.620,-121.289,-37.765,179.090,5.495,149.237
C02452=1203.615,-121.040,-37.774,179.092,5.496,149.236
C02453=1203.610,-120.790,-37.784,179.094,5.496,149.236
C02454=1203.605,-120.539,-37.793,179.096,5.495,149.235
C02455=1203.600,-120.290,-37.803,179.099,5.496,149.235
C02456=1203.594,-120.040,-37.812,179.100,5.496,149.234
C02457=1203.589,-119.790,-37.821,179.103,5.496,149.233
C02458=1203.584,-119.541,-37.831,179.105,5.496,149.233
C02459=1203.578,-119.291,-37.840,179.107,5.497,149.232
C02460=1203.573,-119.041,-37.850,179.109,5.496,149.231
C02461=1203.568,-118.792,-37.859,179.112,5.497,149.231
C02462=1203.562,-118.541,-37.868,179.114,5.497,149.230
C02463=1203.557,-118.292,-37.878,179.116,5.497,149.230
C02464=1203.552,-118.042,-37.887,179.118,5.497,149.229
C02465=1203.546,-117.793,-37.897,179.121,5.497,149.228
C02466=1203.541,-117.543,-37.906,179.123,5.497,149.228
C02467=1203.535,-117.293,-37.915,179.125,5.498,149.227
C02468=1203.530,-117.044,-37.925,179.127,5.497,149.226
C02469=1203.525,-116.794,-37.934,179.130,5.498,149.226
C02470=1203.520,-116.543,-37.944,179.131,5.498,149.225
C02471=1203.515,-116.294,-37.953,179.134,5.498,149.224
C02472=1203.509,-116.044,-37.964,179.136,5.498,149.224
C02473=1203.504,-115.794,-37.972,179.138,5.499,149.223
C02474=1203.499,-115.545,-37.983,179.140,5.498,149.223
C02475=1203.493,-115.295,-37.992,179.142,5.498,149.222
C02476=1203.488,-115.045,-38.002,179.145,5.499,149.221
C02477=1203.483,-114.795,-38.011,179.147,5.498,149.221
C02478=1203.478,-114.546,-38.020,179.149,5.499,149.220
C02479=1203.472,-114.296,-38.030,179.151,5.499,149.219
C02480=1203.468,-114.046,-38.040,179.154,5.499,149.219
C02481=1203.462,-113.796,-38.049,179.156,5.499,149.218
C02482=1203.457,-113.547,-38.059,179.158,5.499,149.218
C02483=1203.451,-113.297,-38.068,179.160,5.499,149.217
C02484=1203.446,-113.047,-38.078,179.163,5.499,149.216
C02485=1203.440,-112.797,-38.087,179.165,5.499,149.215
C02486=1203.435,-112.548,-38.097,179.167,5.500,149.215
C02487=1203.429,-112.298,-38.107,179.169,5.499,149.214
C02488=1203.425,-112.048,-38.116,179.172,5.500,149.213
C02489=1203.420,-111.798,-38.127,179.173,5.500,149.213
C02490=1203.414,-111.548,-38.136,179.176,5.500,149.212
C02491=1203.409,-111.299,-38.146,179.178,5.500,149.212
C02492=1203.404,-111.049,-38.155,179.180,5.501,149.211
C02493=1203.398,-110.800,-38.165,179.182,5.500,149.210
C02494=1203.393,-110.549,-38.175,179.185,5.501,149.210
C02495=1203.388,-110.299,-38.184,179.187,5.501,149.209
C02496=1203.382,-110.050,-38.195,179.189,5.501,149.208
C02497=1203.377,-109.800,-38.203,179.191,5.501,149.208
C02498=1203.372,-109.550,-38.214,179.194,5.501,149.207
C02499=1203.367,-109.301,-38.223,179.196,5.501,149.207
C02500=1203.361,-109.050,-38.233,179.198,5.501,149.206
C02501=1203.357,-108.801,-38.243,179.200,5.501,149.205
C02502=1203.351,-108.552,-38.253,179.203,5.502,149.205
C02503=1203.345,-108.301,-38.262,179.205,5.501,149.204
C02504=1203.340,-108.052,-38.272,179.207,5.502,149.203
C02505=1203.335,-107.802,-38.283,179.209,5.502,149.203
C02506=1203.330,-107.552,-38.292,179.212,5.502,149.202
C02507=1203.324,-107.303,-38.302,179.214,5.502,149.201
C02508=1203.319,-107.053,-38.312,179.216,5.503,149.201
C02509=1203.314,-106.804,-38.322,179.218,5.502,149.200
C02510=1203.309,-106.553,-38.331,179.221,5.503,149.199
C02511=1203.304,-106.304,-38.341,179.223,5.502,149.199
C02512=1203.298,-106.054,-38.351,179.225,5.503,149.198
C02513=1203.292,-105.804,-38.361,179.227,5.503,149.197
C02514=1203.288,-105.554,-38.371,179.230,5.503,149.197
C02515=1203.282,-105.305,-38.381,179.231,5.503,149.196
C02516=1203.277,-105.055,-38.391,179.234,5.504,149.196
C02517=1203.272,-104.806,-38.401,179.236,5.503,149.195
C02518=1203.266,-104.556,-38.410,179.239,5.504,149.194
C02519=1203.261,-104.305,-38.421,179.240,5.504,149.194
C02520=1203.256,-104.056,-38.430,179.243,5.504,149.193
C02521=1203.251,-103.807,-38.441,179.245,5.504,149.192
C02522=1203.245,-103.556,-38.450,179.247,5.504,149.192
C02523=1203.240,-103.306,-38.460,179.249,5.504,149.191
C02524=1203.235,-103.057,-38.470,179.252,5.504,149.190
C02525=1203.229,-102.807,-38.481,179.254,5.504,149.190
C02526=1203.225,-102.557,-38.491,179.256,5.505,149.189
C02527=1203.219,-102.308,-38.501,179.258,5.504,149.188
C02528=1203.213,-102.058,-38.510,179.261,5.505,149.188
C02529=1203.209,-101.809,-38.520,179.263,5.505,149.187
C02530=1203.203,-101.537,-38.531,179.265,5.505,149.186
C02531=1203.198,-101.266,-38.542,179.268,5.506,149.186
C02532=1203.192,-100.994,-38.553,179.270,5.505,149.185
C02533=1203.185,-100.723,-38.564,179.273,5.506,149.184
C02534=1203.180,-100.473,-38.574,179.275,5.505,149.184
C02535=1203.176,-100.223,-38.584,179.278,5.506,149.183
C02536=1203.170,-99.974,-38.594,179.280,5.507,149.182
C02537=1203.165,-99.724,-38.605,179.282,5.506,149.182
C02538=1203.159,-99.474,-38.615,179.285,5.507,149.181
C02539=1203.155,-99.225,-38.625,179.287,5.506,149.180
C02540=1203.149,-98.975,-38.635,179.289,5.507,149.180
C02541=1203.144,-98.725,-38.645,179.291,5.507,149.179
C02542=1203.138,-98.475,-38.656,179.294,5.507,149.178
C02543=1203.133,-98.226,-38.664,179.296,5.507,149.178
C02544=1203.128,-97.975,-38.675,179.298,5.507,149.177
C02545=1203.123,-97.726,-38.685,179.300,5.507,149.176
C02546=1203.117,-97.476,-38.695,179.303,5.507,149.176
C02547=1203.112,-97.226,-38.706,179.305,5.507,149.175
C02548=1203.107,-96.977,-38.716,179.307,5.508,149.175
C02549=1203.102,-96.727,-38.726,179.309,5.507,149.174
C02550=1203.097,-96.477,-38.736,179.312,5.508,149.173
C02551=1203.091,-96.227,-38.747,179.314,5.508,149.172
C02552=1203.085,-95.978,-38.757,179.316,5.508,149.172
C02553=1203.081,-95.728,-38.767,179.318,5.508,149.171
C02554=1203.076,-95.478,-38.777,179.321,5.508,149.171
C02555=1203.071,-95.228,-38.788,179.323,5.509,149.170
C02556=1203.065,-94.979,-38.798,179.325,5.509,149.169
C02557=1203.059,-94.729,-38.808,179.328,5.509,149.169
C02558=1203.054,-94.479,-38.819,179.330,5.509,149.168
C02559=1203.049,-94.229,-38.829,179.332,5.510,149.167
C02560=1203.044,-93.980,-38.838,179.334,5.509,149.167
C02561=1203.039,-93.730,-38.850,179.337,5.510,149.166
C02562=1203.034,-93.481,-38.860,179.339,5.509,149.165
C02563=1203.029,-93.231,-38.870,179.341,5.510,149.165
C02564=1203.023,-92.981,-38.881,179.343,5.510,149.164
C02565=1203.017,-92.732,-38.891,179.346,5.510,149.163
C02566=1203.012,-92.481,-38.901,179.348,5.510,149.163
C02567=1203.007,-92.232,-38.912,179.350,5.510,149.162
C02568=1203.003,-91.982,-38.922,179.352,5.510,149.161
C02569=1202.997,-91.732,-38.932,179.355,5.511,149.161
C02570=1202.991,-91.483,-38.942,179.357,5.511,149.160
C02571=1202.987,-91.233,-38.953,179.359,5.511,149.159
C02572=1202.981,-90.984,-38.964,179.362,5.511,149.159
C02573=1202.976,-90.733,-38.974,179.364,5.511,149.158
C02574=1202.970,-90.484,-38.984,179.366,5.511,149.157
C02575=1202.965,-90.234,-38.995,179.369,5.511,149.157
C02576=1202.960,-89.984,-39.005,179.371,5.512,149.156
C02577=1202.954,-89.734,-39.015,179.373,5.512,149.156
C02578=1202.950,-89.485,-39.027,179.375,5.512,149.155
C02579=1202.944,-89.235,-39.037,179.378,5.512,149.154
C02580=1202.939,-88.985,-39.047,179.380,5.512,149.154
C02581=1202.933,-88.735,-39.058,179.382,5.513,149.153
C02582=1202.928,-88.485,-39.068,179.384,5.512,149.152
C02583=1202.923,-88.236,-39.079,179.387,5.513,149.151
C02584=1202.918,-87.986,-39.090,179.389,5.513,149.151
C02585=1202.913,-87.737,-39.099,179.391,5.513,149.150
C02586=1202.908,-87.487,-39.110,179.394,5.513,149.150
C02587=1202.903,-87.238,-39.121,179.396,5.513,149.149
C02588=1202.897,-86.988,-39.131,179.398,5.513,149.148
C02589=1202.892,-86.738,-39.142,179.400,5.514,149.148
C02590=1202.887,-86.488,-39.152,179.403,5.513,149.147
C02591=1202.882,-86.239,-39.163,179.405,5.514,149.146
C02592=1202.876,-85.989,-39.173,179.408,5.514,149.146
C02593=1202.871,-85.739,-39.184,179.409,5.514,149.145
C02594=1202.865,-85.489,-39.195,179.412,5.515,149.144
C02595=1202.860,-85.239,-39.206,179.414,5.514,149.144
C02596=1202.855,-84.990,-39.216,179.417,5.515,149.143
C02597=1202.850,-84.740,-39.227,179.419,5.515,149.142
C02598=1202.845,-84.491,-39.238,179.421,5.515,149.142
C02599=1202.840,-84.240,-39.248,179.424,5.516,149.141
C02600=1202.834,-83.991,-39.258,179.426,5.515,149.140
C02601=1202.829,-83.741,-39.270,179.429,5.516,149.140
C02602=1202.824,-83.492,-39.280,179.430,5.516,149.139
C02603=1202.819,-83.242,-39.291,179.433,5.516,149.138
C02604=1202.814,-82.992,-39.302,179.435,5.516,149.138
C02605=1202.808,-82.742,-39.312,179.438,5.516,149.137
C02606=1202.803,-82.492,-39.323,179.439,5.516,149.137
C02607=1202.798,-82.243,-39.334,179.442,5.517,149.136
C02608=1202.793,-81.993,-39.344,179.445,5.517,149.135
C02609=1202.788,-81.744,-39.355,179.447,5.517,149.134
C02610=1202.782,-81.493,-39.366,179.449,5.517,149.134
C02611=1202.776,-81.244,-39.376,179.451,5.517,149.133
C02612=1202.772,-80.994,-39.388,179.454,5.517,149.133
C02613=1202.766,-80.745,-39.398,179.456,5.517,149.132
C02614=1202.761,-80.495,-39.409,179.458,5.518,149.131
C02615=1202.756,-80.245,-39.420,179.461,5.518,149.130
C02616=1202.751,-79.996,-39.431,179.463,5.518,149.130
C02617=1202.746,-79.746,-39.441,179.465,5.518,149.129
C02618=1202.740,-79.496,-39.452,179.467,5.518,149.128
C02619=1202.735,-79.246,-39.463,179.470,5.518,149.128
C02620=1202.730,-78.997,-39.474,179.472,5.518,149.127
C02621=1202.725,-78.747,-39.485,179.474,5.519,149.127
C02622=1202.720,-78.497,-39.495,179.477,5.519,149.126
C02623=1202.715,-78.248,-39.506,179.479,5.519,149.125
C02624=1202.709,-77.997,-39.518,179.482,5.519,149.124
C02625=1202.704,-77.748,-39.528,179.483,5.519,149.124
C02626=1202.699,-77.498,-39.539,179.486,5.520,149.123
C02627=1202.694,-77.249,-39.550,179.488,5.519,149.123
C02628=1202.688,-76.999,-39.561,179.491,5.520,149.122
C02629=1202.683,-76.749,-39.572,179.493,5.520,149.121
C02630=1202.677,-76.500,-39.583,179.495,5.520,149.121
C02631=1202.673,-76.250,-39.594,179.498,5.521,149.120
C02632=1202.668,-76.000,-39.605,179.500,5.520,149.119
C02633=1202.662,-75.751,-39.615,179.503,5.521,149.119
C02634=1202.657,-75.480,-39.628,179.505,5.521,149.118
C02635=1202.650,-75.209,-39.640,179.507,5.521,149.117
C02636=1202.645,-74.939,-39.652,179.510,5.521,149.116
C02637=1202.640,-74.668,-39.663,179.513,5.522,149.116
C02638=1202.634,-74.418,-39.674,179.515,5.521,149.115
C02639=1202.629,-74.168,-39.686,179.517,5.522,149.114
C02640=1202.624,-73.919,-39.697,179.520,5.523,149.114
C02641=1202.618,-73.669,-39.708,179.522,5.522,149.113
C02642=1202.613,-73.419,-39.719,179.524,5.523,149.112
C02643=1202.608,-73.169,-39.729,179.526,5.522,149.112
C02644=1202.603,-72.920,-39.740,179.529,5.523,149.111
C02645=1202.597,-72.670,-39.752,179.531,5.524,149.110
C02646=1202.592,-72.420,-39.763,179.533,5.523,149.110
C02647=1202.587,-72.171,-39.774,179.536,5.524,149.109
C02648=1202.582,-71.921,-39.786,179.538,5.523,149.108
C02649=1202.577,-71.671,-39.796,179.541,5.524,149.108
C02650=1202.571,-71.422,-39.807,179.543,5.525,149.107
C02651=1202.566,-71.172,-39.819,179.545,5.524,149.106
C02652=1202.561,-70.922,-39.830,179.548,5.525,149.106
C02653=1202.556,-70.673,-39.841,179.550,5.524,149.105
C02654=1202.551,-70.423,-39.852,179.552,5.525,149.104
C02655=1202.546,-70.173,-39.864,179.555,5.525,149.104
C02656=1202.540,-69.924,-39.874,179.557,5.525,149.103
C02657=1202.535,-69.674,-39.886,179.559,5.526,149.102
C02658=1202.530,-69.424,-39.897,179.561,5.525,149.102
C02659=1202.525,-69.174,-39.908,179.564,5.526,149.101
C02660=1202.519,-68.925,-39.919,179.566,5.526,149.101
C02661=1202.514,-68.675,-39.931,179.568,5.526,149.100
C02662=1202.509,-68.425,-39.942,179.571,5.527,149.099
C02663=1202.503,-68.176,-39.953,179.573,5.526,149.098
C02664=1202.498,-67.926,-39.964,179.576,5.527,149.098
C02665=1202.493,-67.676,-39.976,179.578,5.527,149.097
C02666=1202.488,-67.426,-39.987,179.580,5.527,149.097
C02667=1202.483,-67.177,-39.998,179.583,5.528,149.096
C02668=1202.478,-66.927,-40.010,179.585,5.527,149.095
C02669=1202.473,-66.677,-40.020,179.588,5.528,149.094
C02670=1202.467,-66.427,-40.032,179.590,5.528,149.094
C02671=1202.462,-66.178,-40.043,179.592,5.528,149.093
C02672=1202.457,-65.929,-40.055,179.594,5.528,149.093
C02673=1202.452,-65.679,-40.066,179.597,5.529,149.092
C02674=1202.447,-65.429,-40.078,179.599,5.529,149.091
C02675=1202.441,-65.179,-40.089,179.602,5.529,149.090
C02676=1202.436,-64.930,-40.100,179.604,5.529,149.090
C02677=1202.431,-64.680,-40.112,179.606,5.529,149.089
C02678=1202.426,-64.430,-40.123,179.609,5.530,149.089
C02679=1202.421,-64.181,-40.134,179.611,5.530,149.088
C02680=1202.415,-63.931,-40.146,179.614,5.530,149.087
C02681=1202.410,-63.682,-40.157,179.616,5.530,149.086
C02682=1202.405,-63.432,-40.169,179.618,5.530,149.086
C02683=1202.400,-63.181,-40.180,179.620,5.531,149.085
C02684=1202.395,-62.932,-40.191,179.623,5.531,149.085
C02685=1202.389,-62.683,-40.202,179.625,5.531,149.084
C02686=1202.384,-62.433,-40.214,179.628,5.531,149.083
C02687=1202.379,-62.183,-40.226,179.630,5.531,149.082
C02688=1202.374,-61.933,-40.237,179.632,5.532,149.082
C02689=1202.369,-61.683,-40.249,179.635,5.532,149.081
C02690=1202.363,-61.434,-40.260,179.637,5.532,149.081
C02691=1202.358,-61.185,-40.272,179.640,5.532,149.080
C02692=1202.353,-60.935,-40.283,179.642,5.532,149.079
C02693=1202.348,-60.685,-40.295,179.644,5.533,149.079
C02694=1202.343,-60.435,-40.307,179.647,5.533,149.078
C02695=1202.338,-60.185,-40.318,179.649,5.533,149.077
C02696=1202.332,-59.936,-40.329,179.651,5.533,149.077
C02697=1202.327,-59.686,-40.341,179.654,5.534,149.076
C02698=1202.322,-59.437,-40.353,179.656,5.533,149.075
C02699=1202.317,-59.187,-40.364,179.658,5.534,149.075
C02700=1202.312,-58.937,-40.376,179.661,5.535,149.074
C02701=1202.306,-58.687,-40.388,179.663,5.534,149.073
C02702=1202.302,-58.438,-40.399,179.666,5.535,149.073
C02703=1202.296,-58.188,-40.410,179.668,5.534,149.072
C02704=1202.291,-57.939,-40.422,179.670,5.535,149.071
C02705=1202.286,-57.689,-40.434,179.673,5.536,149.071
C02706=1202.280,-57.439,-40.446,179.675,5.535,149.070
C02707=1202.276,-57.190,-40.458,179.677,5.536,149.069
C02708=1202.270,-56.940,-40.469,179.680,5.536,149.069
C02709=1202.266,-56.690,-40.481,179.682,5.536,149.068
C02710=1202.260,-56.440,-40.493,179.685,5.536,149.067
C02711=1202.255,-56.190,-40.504,179.687,5.537,149.067
C02712=1202.250,-55.941,-40.515,179.689,5.537,149.066
C02713=1202.244,-55.692,-40.527,179.692,5.537,149.065
C02714=1202.239,-55.442,-40.539,179.694,5.538,149.065
C02715=1202.234,-55.193,-40.551,179.696,5.537,149.064
C02716=1202.229,-54.943,-40.563,179.699,5.538,149.063
C02717=1202.224,-54.693,-40.574,179.701,5.539,149.063
C02718=1202.219,-54.443,-40.586,179.703,5.538,149.062
C02719=1202.213,-54.193,-40.598,179.706,5.539,149.061
C02720=1202.209,-53.944,-40.610,179.708,5.538,149.061
C02721=1202.203,-53.694,-40.622,179.711,5.539,149.060
C02722=1202.198,-53.444,-40.634,179.713,5.539,149.059
C02723=1202.193,-53.195,-40.645,179.715,5.539,149.059
C02724=1202.188,-52.945,-40.657,179.718,5.540,149.058
C02725=1202.183,-52.695,-40.670,179.720,5.540,149.057
C02726=1202.177,-52.446,-40.681,179.722,5.540,149.057
C02727=1202.172,-52.197,-40.692,179.725,5.540,149.056
C02728=1202.167,-51.947,-40.704,179.728,5.541,149.055
C02729=1202.161,-51.697,-40.716,179.729,5.541,149.055
C02730=1202.157,-51.448,-40.728,179.732,5.541,149.054
C02731=1202.151,-51.198,-40.740,179.735,5.542,149.053
C02732=1202.146,-50.948,-40.752,179.737,5.541,149.053
C02733=1202.141,-50.698,-40.765,179.739,5.542,149.052
C02734=1202.136,-50.449,-40.776,179.742,5.542,149.051
C02735=1202.131,-50.199,-40.788,179.744,5.542,149.051
C02736=1202.125,-49.949,-40.800,179.746,5.543,149.050
C02737=1202.120,-49.700,-40.812,179.749,5.543,149.049
C02738=1202.115,-49.429,-40.825,179.752,5.544,149.049
C02739=1202.109,-49.160,-40.838,179.754,5.543,149.048
C02740=1202.104,-48.889,-40.851,179.756,5.544,149.047
C02741=1202.098,-48.619,-40.864,179.759,5.544,149.046
C02742=1202.093,-48.369,-40.876,179.762,5.545,149.046
C02743=1202.088,-48.120,-40.888,179.764,5.544,149.045
C02744=1202.083,-47.870,-40.900,179.767,5.545,149.044
C02745=1202.078,-47.620,-40.911,179.769,5.545,149.044
C02746=1202.073,-47.371,-40.924,179.771,5.545,149.043
C02747=1202.067,-47.121,-40.936,179.773,5.546,149.042
C02748=1202.062,-46.872,-40.949,179.776,5.546,149.042
C02749=1202.057,-46.622,-40.960,179.778,5.546,149.041
C02750=1202.052,-46.372,-40.972,179.781,5.546,149.040
C02751=1202.047,-46.123,-40.984,179.784,5.547,149.040
C02752=1202.041,-45.873,-40.996,179.786,5.546,149.039
C02753=1202.036,-45.623,-41.009,179.788,5.547,149.038
C02754=1202.031,-45.373,-41.021,179.790,5.548,149.038
C02755=1202.026,-45.124,-41.033,179.793,5.548,149.037
C02756=1202.021,-44.875,-41.045,179.795,5.548,149.036
C02757=1202.015,-44.625,-41.056,179.798,5.548,149.036
C02758=1202.010,-44.375,-41.069,179.801,5.549,149.035
C02759=1202.005,-44.125,-41.081,179.803,5.548,149.034
C02760=1202.000,-43.876,-41.094,179.805,5.549,149.034
C02761=1201.994,-43.626,-41.105,179.807,5.550,149.033
C02762=1201.989,-43.377,-41.118,179.810,5.549,149.032
C02763=1201.984,-43.127,-41.130,179.812,5.550,149.032
C02764=1201.980,-42.877,-41.142,179.815,5.550,149.031
C02765=1201.975,-42.627,-41.154,179.817,5.550,149.030
C02766=1201.970,-42.378,-41.167,179.820,5.550,149.030
C02767=1201.964,-42.128,-41.179,179.822,5.551,149.029
C02768=1201.959,-41.879,-41.191,179.824,5.552,149.028
C02769=1201.954,-41.629,-41.204,179.826,5.551,149.028
C02770=1201.948,-41.379,-41.216,179.829,5.552,149.027
C02771=1201.943,-41.130,-41.228,179.832,5.552,149.026
C02772=1201.938,-40.880,-41.240,179.834,5.552,149.026
C02773=1201.933,-40.631,-41.253,179.836,5.553,149.025
C02774=1201.928,-40.380,-41.265,179.839,5.553,149.024
C02775=1201.923,-40.131,-41.278,179.841,5.553,149.024
C02776=1201.918,-39.882,-41.290,179.843,5.553,149.023
C02777=1201.912,-39.632,-41.302,179.846,5.554,149.022
C02778=1201.907,-39.382,-41.315,179.849,5.554,149.022
C02779=1201.902,-39.132,-41.327,179.851,5.554,149.021
C02780=1201.897,-38.883,-41.339,179.853,5.555,149.020
C02781=1201.891,-38.634,-41.352,179.856,5.555,149.020
C02782=1201.887,-38.383,-41.364,179.858,5.555,149.019
C02783=1201.881,-38.134,-41.377,179.860,5.555,149.018
C02784=1201.876,-37.884,-41.389,179.863,5.556,149.018
C02785=1201.871,-37.634,-41.401,179.866,5.556,149.017
C02786=1201.866,-37.385,-41.414,179.867,5.556,149.017
C02787=1201.861,-37.136,-41.426,179.870,5.557,149.016
C02788=1201.855,-36.886,-41.438,179.873,5.557,149.015
C02789=1201.851,-36.636,-41.451,179.875,5.557,149.014
C02790=1201.846,-36.387,-41.464,179.877,5.557,149.014
C02791=1201.840,-36.137,-41.476,179.880,5.558,149.013
C02792=1201.835,-35.887,-41.488,179.883,5.558,149.012
C02793=1201.830,-35.638,-41.501,179.884,5.558,149.012
C02794=1201.825,-35.388,-41.514,179.887,5.559,149.011
C02795=1201.820,-35.138,-41.526,179.890,5.559,149.010
C02796=1201.815,-34.889,-41.538,179.892,5.559,149.010
C02797=1201.810,-34.639,-41.551,179.894,5.559,149.009
C02798=1201.805,-34.390,-41.564,179.897,5.560,149.008
C02799=1201.800,-34.139,-41.576,179.899,5.561,149.008
C02800=1201.794,-33.890,-41.589,179.901,5.560,149.007
C02801=1201.789,-33.641,-41.602,179.904,5.561,149.006
C02802=1201.784,-33.391,-41.614,179.907,5.561,149.006
C02803=1201.778,-33.141,-41.626,179.909,5.562,149.005
C02804=1201.774,-32.891,-41.639,179.911,5.561,149.004
C02805=1201.769,-32.642,-41.652,179.914,5.562,149.004
C02806=1201.763,-32.393,-41.664,179.916,5.563,149.003
C02807=1201.758,-32.143,-41.677,179.919,5.563,149.003
C02808=1201.752,-31.894,-41.690,179.921,5.563,149.002
C02809=1201.748,-31.643,-41.702,179.924,5.563,149.001
C02810=1201.743,-31.394,-41.715,179.926,5.564,149.000
C02811=1201.737,-31.144,-41.728,179.928,5.563,149.000
C02812=1201.732,-30.895,-41.740,179.931,5.564,148.999
C02813=1201.728,-30.645,-41.753,179.933,5.565,148.999
C02814=1201.723,-30.396,-41.766,179.936,5.565,148.998
C02815=1201.717,-30.146,-41.779,179.938,5.565,148.997
C02816=1201.712,-29.896,-41.792,179.941,5.565,148.996
C02817=1201.707,-29.646,-41.804,179.943,5.566,148.996
C02818=1201.702,-29.397,-41.816,179.946,5.566,148.995
C02819=1201.697,-29.148,-41.829,179.948,5.566,148.995
C02820=1201.691,-28.897,-41.842,179.950,5.567,148.994
C02821=1201.686,-28.648,-41.855,179.953,5.567,148.993
C02822=1201.681,-28.399,-41.868,179.956,5.568,148.993
C02823=1201.676,-28.149,-41.880,179.958,5.567,148.992
C02824=1201.671,-27.899,-41.893,179.960,5.568,148.991
C02825=1201.666,-27.650,-41.906,179.963,5.568,148.990
C02826=1201.660,-27.400,-41.919,179.965,5.569,148.990
C02827=1201.656,-27.150,-41.932,179.967,5.569,148.989
C02828=1201.651,-26.901,-41.945,179.970,5.569,148.989
C02829=1201.645,-26.651,-41.958,179.973,5.570,148.988
C02830=1201.640,-26.401,-41.971,179.975,5.570,148.987
C02831=1201.635,-26.152,-41.983,179.977,5.570,148.986
C02832=1201.630,-25.903,-41.996,179.980,5.570,148.986
C02833=1201.625,-25.652,-42.010,179.982,5.571,148.985
C02834=1201.620,-25.403,-42.022,179.985,5.572,148.985
C02835=1201.615,-25.154,-42.035,179.987,5.572,148.984
C02836=1201.609,-24.903,-42.048,179.989,5.572,148.983
C02837=1201.604,-24.654,-42.061,179.992,5.572,148.983
C02838=1201.599,-24.405,-42.074,179.995,5.573,148.982
C02839=1201.595,-24.155,-42.086,179.997,5.574,148.981
C02840=1201.589,-23.905,-42.100,179.999,5.573,148.981
C02841=1201.584,-23.656,-42.113,-179.998,5.574,148.980
C02842=1201.578,-23.386,-42.127,-179.996,5.574,148.979
C02843=1201.573,-23.117,-42.141,-179.993,5.575,148.979
C02844=1201.567,-22.847,-42.155,-179.990,5.575,148.978
C02845=1201.562,-22.578,-42.169,-179.988,5.576,148.977
C02846=1201.557,-22.328,-42.183,-179.985,5.576,148.976
C02847=1201.552,-22.079,-42.195,-179.983,5.576,148.976
C02848=1201.547,-21.829,-42.208,-179.980,5.576,148.975
C02849=1201.541,-21.579,-42.222,-179.978,5.577,148.974
C02850=1201.536,-21.330,-42.234,-179.975,5.577,148.974
C02851=1201.531,-21.080,-42.247,-179.973,5.577,148.973
C02852=1201.526,-20.830,-42.260,-179.971,5.578,148.973
C02853=1201.521,-20.581,-42.274,-179.968,5.578,148.972
C02854=1201.516,-20.331,-42.287,-179.965,5.579,148.971
C02855=1201.511,-20.082,-42.300,-179.963,5.579,148.970
C02856=1201.506,-19.832,-42.312,-179.961,5.579,148.970
C02857=1201.500,-19.582,-42.326,-179.958,5.579,148.969
C02858=1201.495,-19.333,-42.339,-179.955,5.580,148.968
C02859=1201.490,-19.083,-42.353,-179.953,5.581,148.968
C02860=1201.485,-18.834,-42.365,-179.951,5.580,148.967
C02861=1201.481,-18.584,-42.378,-179.948,5.581,148.967
C02862=1201.475,-18.335,-42.392,-179.946,5.581,148.966
C02863=1201.470,-18.085,-42.405,-179.943,5.582,148.965
C02864=1201.465,-17.835,-42.419,-179.940,5.582,148.964
C02865=1201.459,-17.586,-42.431,-179.939,5.582,148.964
C02866=1201.455,-17.336,-42.445,-179.936,5.583,148.963
C02867=1201.449,-17.087,-42.458,-179.934,5.583,148.963
C02868=1201.444,-16.836,-42.472,-179.931,5.584,148.962
C02869=1201.439,-16.588,-42.485,-179.928,5.584,148.961
C02870=1201.434,-16.337,-42.498,-179.926,5.584,148.960
C02871=1201.429,-16.088,-42.511,-179.923,5.584,148.960
C02872=1201.423,-15.839,-42.525,-179.921,5.585,148.959
C02873=1201.419,-15.589,-42.538,-179.919,5.586,148.959
C02874=1201.413,-15.339,-42.551,-179.916,5.586,148.958
C02875=1201.409,-15.090,-42.565,-179.914,5.586,148.957
C02876=1201.403,-14.840,-42.578,-179.911,5.586,148.957
C02877=1201.398,-14.590,-42.591,-179.909,5.587,148.956
C02878=1201.393,-14.341,-42.605,-179.906,5.588,148.955
C02879=1201.388,-14.091,-42.618,-179.904,5.588,148.955
C02880=1201.383,-13.842,-42.632,-179.902,5.588,148.954
C02881=1201.378,-13.592,-42.645,-179.899,5.588,148.953
C02882=1201.372,-13.342,-42.658,-179.896,5.589,148.953
C02883=1201.368,-13.093,-42.672,-179.894,5.589,148.952
C02884=1201.362,-12.843,-42.685,-179.891,5.590,148.951
C02885=1201.358,-12.594,-42.698,-179.889,5.590,148.951
C02886=1201.352,-12.344,-42.712,-179.887,5.590,148.950
C02887=1201.347,-12.094,-42.725,-179.884,5.591,148.949
C02888=1201.342,-11.845,-42.739,-179.882,5.591,148.949
C02889=1201.337,-11.595,-42.752,-179.879,5.592,148.948
C02890=1201.333,-11.346,-42.766,-179.876,5.592,148.947
C02891=1201.327,-11.096,-42.779,-179.875,5.592,148.947
C02892=1201.323,-10.847,-42.793,-179.872,5.593,148.946
C02893=1201.317,-10.597,-42.806,-179.869,5.593,148.945
C02894=1201.312,-10.347,-42.820,-179.867,5.594,148.945
C02895=1201.307,-10.098,-42.833,-179.864,5.594,148.944
C02896=1201.302,-9.848,-42.847,-179.861,5.595,148.943
C02897=1201.296,-9.599,-42.860,-179.860,5.595,148.943
C02898=1201.292,-9.349,-42.874,-179.857,5.595,148.942
C02899=1201.286,-9.099,-42.887,-179.854,5.596,148.942
C02900=1201.282,-8.850,-42.901,-179.852,5.596,148.941
C02901=1201.277,-8.601,-42.915,-179.849,5.597,148.940
C02902=1201.271,-8.351,-42.928,-179.846,5.597,148.939
C02903=1201.267,-8.101,-42.942,-179.844,5.597,148.939
C02904=1201.261,-7.852,-42.955,-179.842,5.598,148.938
C02905=1201.256,-7.602,-42.969,-179.840,5.598,148.938
C02906=1201.251,-7.353,-42.983,-179.837,5.599,148.937
C02907=1201.246,-7.103,-42.996,-179.834,5.599,148.936
C02908=1201.241,-6.853,-43.011,-179.832,5.600,148.936
C02909=1201.236,-6.604,-43.023,-179.830,5.599,148.935
C02910=1201.231,-6.354,-43.037,-179.827,5.600,148.934
C02911=1201.226,-6.105,-43.052,-179.825,5.601,148.934
C02912=1201.220,-5.855,-43.065,-179.822,5.601,148.933
C02913=1201.216,-5.606,-43.079,-179.819,5.602,148.932
C02914=1201.211,-5.356,-43.093,-179.817,5.602,148.932
C02915=1201.205,-5.106,-43.106,-179.815,5.602,148.931
C02916=1201.201,-4.857,-43.120,-179.813,5.603,148.930
C02917=1201.195,-4.608,-43.134,-179.810,5.603,148.930
C02918=1201.190,-4.358,-43.147,-179.807,5.604,148.929
C02919=1201.185,-4.108,-43.161,-179.805,5.604,148.928
C02920=1201.180,-3.859,-43.175,-179.802,5.605,148.928
C02921=1201.175,-3.609,-43.188,-179.799,5.605,148.927
C02922=1201.170,-3.359,-43.203,-179.798,5.605,148.927
C02923=1201.164,-3.110,-43.217,-179.795,5.606,148.926
C02924=1201.159,-2.860,-43.231,-179.792,5.606,148.925
C02925=1201.155,-2.610,-43.244,-179.790,5.607,148.924
C02926=1201.149,-2.361,-43.258,-179.787,5.607,148.924
C02927=1201.144,-2.112,-43.272,-179.784,5.608,148.923
C02928=1201.139,-1.862,-43.286,-179.782,5.608,148.923
C02929=1201.134,-1.613,-43.299,-179.780,5.608,148.922
C02930=1201.129,-1.363,-43.313,-179.777,5.609,148.921
C02931=1201.124,-1.113,-43.327,-179.775,5.609,148.921
C02932=1201.119,-0.864,-43.341,-179.772,5.610,148.920
C02933=1201.114,-0.614,-43.356,-179.770,5.610,148.919
C02934=1201.108,-0.364,-43.369,-179.767,5.611,148.919
C02935=1201.104,-0.115,-43.383,-179.765,5.611,148.918
C02936=1201.099,0.134,-43.397,-179.762,5.612,148.917
C02937=1201.094,0.384,-43.411,-179.760,5.612,148.917
C02938=1201.089,0.634,-43.425,-179.757,5.612,148.916
C02939=1201.083,0.883,-43.439,-179.755,5.613,148.915
C02940=1201.078,1.132,-43.453,-179.753,5.613,148.915
C02941=1201.073,1.383,-43.467,-179.750,5.614,148.914
C02942=1201.068,1.632,-43.481,-179.747,5.614,148.913
C02943=1201.063,1.881,-43.495,-179.745,5.615,148.913
C02944=1201.058,2.131,-43.509,-179.742,5.615,148.912
C02945=1201.053,2.381,-43.523,-179.740,5.615,148.911
C02946=1201.048,2.650,-43.538,-179.737,5.616,148.911
C02947=1201.042,2.918,-43.554,-179.735,5.616,148.910
C02948=1201.037,3.187,-43.569,-179.731,5.617,148.909
C02949=1201.031,3.457,-43.584,-179.729,5.618,148.909
C02950=1201.026,3.707,-43.598,-179.727,5.618,148.908
C02951=1201.021,3.956,-43.612,-179.724,5.618,148.908
C02952=1201.016,4.205,-43.626,-179.722,5.619,148.907
C02953=1201.011,4.455,-43.640,-179.719,5.619,148.906
C02954=1201.006,4.705,-43.655,-179.716,5.620,148.905
C02955=1201.001,4.954,-43.669,-179.714,5.620,148.905
C02956=1200.995,5.203,-43.683,-179.711,5.621,148.904
C02957=1200.990,5.453,-43.697,-179.709,5.622,148.904
C02958=1200.985,5.703,-43.711,-179.706,5.622,148.903
C02959=1200.980,5.953,-43.726,-179.704,5.622,148.902
C02960=1200.976,6.202,-43.740,-179.702,5.622,148.902
C02961=1200.970,6.451,-43.754,-179.699,5.623,148.901
C02962=1200.965,6.701,-43.768,-179.696,5.623,148.900
C02963=1200.960,6.951,-43.782,-179.694,5.624,148.900
C02964=1200.955,7.200,-43.797,-179.691,5.625,148.899
C02965=1200.950,7.450,-43.812,-179.689,5.625,148.898
C02966=1200.945,7.699,-43.825,-179.686,5.626,148.898
C02967=1200.940,7.948,-43.840,-179.684,5.626,148.897
C02968=1200.935,8.198,-43.854,-179.681,5.627,148.897
C02969=1200.930,8.448,-43.868,-179.679,5.628,148.896
C02970=1200.925,8.697,-43.883,-179.677,5.627,148.895
C02971=1200.920,8.947,-43.897,-179.674,5.628,148.894
C02972=1200.915,9.196,-43.911,-179.671,5.628,148.894
C02973=1200.910,9.446,-43.925,-179.669,5.629,148.893
C02974=1200.905,9.695,-43.940,-179.667,5.630,148.893
C02975=1200.900,9.945,-43.954,-179.664,5.630,148.892
C02976=1200.895,10.194,-43.969,-179.661,5.631,148.891
C02977=1200.890,10.444,-43.983,-179.659,5.631,148.891
C02978=1200.885,10.694,-43.997,-179.656,5.632,148.890
C02979=1200.879,10.943,-44.012,-179.654,5.633,148.889
C02980=1200.874,11.192,-44.027,-179.651,5.633,148.889
C02981=1200.869,11.442,-44.041,-179.648,5.634,148.888
C02982=1200.864,11.692,-44.055,-179.646,5.633,148.887
C02983=1200.859,11.941,-44.069,-179.644,5.634,148.887
C02984=1200.854,12.191,-44.084,-179.641,5.634,148.886
C02985=1200.850,12.440,-44.099,-179.639,5.635,148.886
C02986=1200.845,12.690,-44.113,-179.636,5.636,148.885
C02987=1200.839,12.940,-44.128,-179.634,5.636,148.884
C02988=1200.834,13.189,-44.142,-179.631,5.637,148.884
C02989=1200.829,13.438,-44.157,-179.628,5.637,148.883
C02990=1200.824,13.688,-44.171,-179.626,5.638,148.882
C02991=1200.819,13.937,-44.185,-179.624,5.639,148.882
C02992=1200.814,14.186,-44.200,-179.621,5.639,148.881
C02993=1200.809,14.436,-44.215,-179.618,5.640,148.880
C02994=1200.804,14.686,-44.230,-179.616,5.640,148.880
C02995=1200.799,14.936,-44.244,-179.613,5.641,148.879
C02996=1200.794,15.185,-44.259,-179.611,5.641,148.879
C02997=1200.789,15.435,-44.273,-179.609,5.641,148.878
C02998=1200.784,15.684,-44.287,-179.606,5.642,148.877
C02999=1200.779,15.934,-44.303,-179.603,5.642,148.876
C03000=1200.774,16.184,-44.317,-179.601,5.643,148.876
C03001=1200.769,16.433,-44.332,-179.599,5.644,148.875
C03002=1200.764,16.682,-44.346,-179.596,5.644,148.875
C03003=1200.758,16.932,-44.361,-179.593,5.645,148.874
C03004=1200.753,17.181,-44.376,-179.591,5.645,148.873
C03005=1200.748,17.430,-44.390,-179.588,5.646,148.873
C03006=1200.743,17.680,-44.405,-179.586,5.647,148.872
C03007=1200.738,17.930,-44.420,-179.583,5.647,148.871
C03008=1200.733,18.179,-44.434,-179.581,5.648,148.871
C03009=1200.728,18.428,-44.449,-179.578,5.648,148.870
C03010=1200.723,18.678,-44.464,-179.576,5.649,148.870
C03011=1200.718,18.927,-44.479,-179.573,5.649,148.869
C03012=1200.713,19.177,-44.494,-179.570,5.650,148.868
C03013=1200.708,19.426,-44.509,-179.568,5.650,148.868
C03014=1200.703,19.676,-44.523,-179.565,5.651,148.867
C03015=1200.698,19.925,-44.538,-179.563,5.652,148.866
C03016=1200.693,20.175,-44.553,-179.560,5.652,148.866
C03017=1200.688,20.424,-44.568,-179.558,5.653,148.865
C03018=1200.683,20.674,-44.583,-179.556,5.653,148.864
C03019=1200.678,20.923,-44.598,-179.553,5.653,148.864
C03020=1200.673,21.173,-44.612,-179.551,5.654,148.863
C03021=1200.668,21.422,-44.627,-179.548,5.654,148.863
C03022=1200.663,21.672,-44.642,-179.546,5.655,148.862
C03023=1200.658,21.921,-44.657,-179.543,5.655,148.861
C03024=1200.653,22.172,-44.672,-179.540,5.656,148.861
C03025=1200.648,22.421,-44.687,-179.538,5.657,148.860
C03026=1200.644,22.671,-44.701,-179.535,5.657,148.859
C03027=1200.638,22.920,-44.717,-179.533,5.658,148.859
C03028=1200.633,23.169,-44.732,-179.530,5.658,148.858
C03029=1200.628,23.419,-44.747,-179.527,5.659,148.857
C03030=1200.623,23.668,-44.762,-179.525,5.660,148.857
C03031=1200.618,23.918,-44.776,-179.523,5.660,148.856
C03032=1200.613,24.167,-44.791,-179.520,5.661,148.856
C03033=1200.608,24.417,-44.806,-179.517,5.661,148.855
C03034=1200.602,24.667,-44.821,-179.515,5.662,148.854
C03035=1200.598,24.916,-44.836,-179.513,5.663,148.854
C03036=1200.593,25.165,-44.851,-179.510,5.663,148.853
C03037=1200.587,25.415,-44.866,-179.507,5.664,148.852
C03038=1200.583,25.664,-44.881,-179.505,5.664,148.852
C03039=1200.578,25.914,-44.897,-179.502,5.665,148.851
C03040=1200.573,26.164,-44.911,-179.500,5.666,148.851
C03041=1200.568,26.413,-44.927,-179.497,5.666,148.850
C03042=1200.563,26.662,-44.942,-179.495,5.667,148.849
C03043=1200.557,26.912,-44.957,-179.492,5.667,148.849
C03044=1200.553,27.161,-44.972,-179.490,5.668,148.848
C03045=1200.547,27.411,-44.987,-179.487,5.669,148.847
C03046=1200.543,27.660,-45.002,-179.484,5.669,148.847
C03047=1200.538,27.911,-45.018,-179.482,5.670,148.846
C03048=1200.533,28.160,-45.033,-179.480,5.671,148.846
C03049=1200.528,28.409,-45.048,-179.477,5.671,148.845
C03050=1200.522,28.678,-45.064,-179.474,5.672,148.844
C03051=1200.517,28.946,-45.081,-179.472,5.672,148.844
C03052=1200.512,29.215,-45.097,-179.468,5.673,148.843
C03053=1200.506,29.484,-45.114,-179.466,5.674,148.842
C03054=1200.501,29.733,-45.128,-179.463,5.674,148.842
C03055=1200.496,29.983,-45.144,-179.461,5.675,148.841
C03056=1200.491,30.232,-45.159,-179.458,5.675,148.840
C03057=1200.486,30.482,-45.175,-179.456,5.676,148.840
C03058=1200.481,30.731,-45.190,-179.453,5.677,148.839
C03059=1200.476,30.980,-45.205,-179.450,5.677,148.838
C03060=1200.471,31.230,-45.220,-179.448,5.678,148.838
C03061=1200.466,31.479,-45.235,-179.446,5.679,148.837
C03062=1200.461,31.730,-45.251,-179.443,5.679,148.837
C03063=1200.457,31.979,-45.266,-179.440,5.680,148.836
C03064=1200.451,32.228,-45.282,-179.438,5.680,148.835
C03065=1200.446,32.477,-45.297,-179.436,5.681,148.835
C03066=1200.441,32.727,-45.312,-179.433,5.682,148.834
C03067=1200.436,32.977,-45.328,-179.430,5.682,148.833
C03068=1200.432,33.226,-45.343,-179.428,5.683,148.833
C03069=1200.426,33.475,-45.359,-179.425,5.683,148.832
C03070=1200.421,33.725,-45.373,-179.423,5.684,148.832
C03071=1200.416,33.974,-45.388,-179.420,5.685,148.831
C03072=1200.411,34.224,-45.404,-179.418,5.685,148.830
C03073=1200.406,34.474,-45.420,-179.415,5.686,148.830
C03074=1200.401,34.723,-45.435,-179.413,5.687,148.829
C03075=1200.396,34.972,-45.451,-179.410,5.687,148.828
C03076=1200.391,35.222,-45.467,-179.407,5.688,148.828
C03077=1200.386,35.471,-45.482,-179.405,5.688,148.827
C03078=1200.381,35.721,-45.497,-179.403,5.689,148.827
C03079=1200.376,35.970,-45.513,-179.400,5.690,148.826
C03080=1200.372,36.220,-45.528,-179.397,5.690,148.825
C03081=1200.366,36.469,-45.544,-179.394,5.691,148.825
C03082=1200.361,36.719,-45.559,-179.392,5.692,148.824
C03083=1200.356,36.967,-45.575,-179.389,5.693,148.824
C03084=1200.352,37.217,-45.591,-179.387,5.693,148.823
C03085=1200.346,37.467,-45.607,-179.384,5.694,148.822
C03086=1200.341,37.716,-45.622,-179.382,5.695,148.822
C03087=1200.336,37.965,-45.637,-179.379,5.695,148.821
C03088=1200.331,38.215,-45.653,-179.377,5.696,148.820
C03089=1200.326,38.465,-45.669,-179.374,5.696,148.820
C03090=1200.321,38.714,-45.684,-179.372,5.697,148.819
C03091=1200.317,38.964,-45.700,-179.369,5.698,148.819
C03092=1200.311,39.213,-45.715,-179.367,5.698,148.818
C03093=1200.306,39.462,-45.731,-179.364,5.699,148.817
C03094=1200.301,39.712,-45.747,-179.362,5.700,148.817
C03095=1200.297,39.961,-45.762,-179.359,5.700,148.816
C03096=1200.291,40.211,-45.778,-179.357,5.701,148.815
C03097=1200.287,40.461,-45.794,-179.354,5.701,148.815
C03098=1200.281,40.710,-45.810,-179.352,5.702,148.814
C03099=1200.276,40.959,-45.826,-179.348,5.704,148.814
C03100=1200.272,41.209,-45.841,-179.346,5.704,148.813
C03101=1200.267,41.458,-45.857,-179.343,5.705,148.812
C03102=1200.261,41.708,-45.872,-179.341,5.706,148.812
C03103=1200.256,41.958,-45.888,-179.338,5.706,148.811
C03104=1200.251,42.207,-45.905,-179.336,5.707,148.811
C03105=1200.247,42.456,-45.920,-179.333,5.707,148.810
C03106=1200.242,42.706,-45.936,-179.331,5.708,148.809
C03107=1200.237,42.955,-45.951,-179.328,5.709,148.809
C03108=1200.231,43.204,-45.967,-179.326,5.709,148.808
C03109=1200.227,43.454,-45.983,-179.323,5.710,148.807
C03110=1200.221,43.703,-45.999,-179.321,5.710,148.807
C03111=1200.216,43.952,-46.015,-179.318,5.711,148.806
C03112=1200.211,44.202,-46.031,-179.315,5.712,148.806
C03113=1200.207,44.451,-46.046,-179.312,5.713,148.805
C03114=1200.202,44.702,-46.062,-179.310,5.714,148.805
C03115=1200.197,44.950,-46.079,-179.308,5.714,148.804
C03116=1200.192,45.200,-46.094,-179.305,5.715,148.803
C03117=1200.187,45.450,-46.110,-179.303,5.716,148.803
C03118=1200.182,45.699,-46.126,-179.300,5.716,148.802
C03119=1200.177,45.949,-46.142,-179.298,5.717,148.801
C03120=1200.172,46.197,-46.159,-179.295,5.717,148.801
C03121=1200.167,46.448,-46.175,-179.293,5.718,148.800
C03122=1200.162,46.697,-46.190,-179.290,5.719,148.800
C03123=1200.157,46.946,-46.206,-179.287,5.720,148.799
C03124=1200.152,47.196,-46.222,-179.284,5.721,148.798
C03125=1200.147,47.444,-46.238,-179.282,5.722,148.798
C03126=1200.143,47.694,-46.254,-179.279,5.722,148.797
C03127=1200.137,47.944,-46.270,-179.277,5.723,148.796
C03128=1200.133,48.193,-46.286,-179.275,5.724,148.796
C03129=1200.127,48.443,-46.302,-179.272,5.724,148.795
C03130=1200.122,48.692,-46.318,-179.269,5.725,148.795
C03131=1200.117,48.942,-46.334,-179.267,5.725,148.794
C03132=1200.112,49.190,-46.350,-179.264,5.727,148.794
C03133=1200.108,49.441,-46.366,-179.261,5.727,148.793
C03134=1200.103,49.689,-46.383,-179.259,5.728,148.792
C03135=1200.098,49.939,-46.399,-179.257,5.729,148.792
C03136=1200.093,50.188,-46.415,-179.254,5.729,148.791
C03137=1200.088,50.438,-46.431,-179.251,5.730,148.790
C03138=1200.083,50.687,-46.447,-179.249,5.730,148.790
C03139=1200.078,50.937,-46.463,-179.247,5.731,148.789
C03140=1200.072,51.186,-46.480,-179.243,5.733,148.789
C03141=1200.067,51.436,-46.496,-179.241,5.733,148.788
C03142=1200.062,51.685,-46.512,-179.239,5.734,148.788
C03143=1200.058,51.935,-46.529,-179.236,5.735,148.787
C03144=1200.052,52.184,-46.545,-179.233,5.735,148.786
C03145=1200.048,52.434,-46.561,-179.231,5.736,148.786
C03146=1200.043,52.683,-46.577,-179.229,5.737,148.785
C03147=1200.038,52.932,-46.594,-179.226,5.737,148.784
C03148=1200.033,53.181,-46.610,-179.223,5.738,148.784
C03149=1200.028,53.431,-46.626,-179.221,5.739,148.783
C03150=1200.024,53.681,-46.642,-179.218,5.740,148.783
C03151=1200.019,53.930,-46.659,-179.215,5.740,148.782
C03152=1200.013,54.180,-46.675,-179.213,5.741,148.781
C03153=1200.008,54.429,-46.692,-179.210,5.742,148.781
C03154=1200.003,54.697,-46.709,-179.207,5.743,148.780
C03155=1199.998,54.966,-46.727,-179.205,5.744,148.780
C03156=1199.992,55.234,-46.744,-179.202,5.744,148.779
C03157=1199.987,55.503,-46.762,-179.199,5.745,148.778
C03158=1199.982,55.752,-46.779,-179.196,5.746,148.778
C03159=1199.977,56.002,-46.795,-179.194,5.747,148.777
C03160=1199.972,56.251,-46.811,-179.191,5.748,148.777
C03161=1199.968,56.500,-46.828,-179.189,5.748,148.776
C03162=1199.962,56.750,-46.843,-179.187,5.749,148.775
C03163=1199.957,57.000,-46.861,-179.184,5.750,148.775
C03164=1199.952,57.249,-46.877,-179.181,5.751,148.774
C03165=1199.947,57.498,-46.894,-179.179,5.752,148.774
C03166=1199.943,57.748,-46.909,-179.176,5.752,148.773
C03167=1199.937,57.997,-46.926,-179.173,5.753,148.772
C03168=1199.932,58.246,-46.943,-179.171,5.754,148.772
C03169=1199.928,58.496,-46.960,-179.169,5.754,148.771
C03170=1199.923,58.745,-46.976,-179.166,5.755,148.771
C03171=1199.918,58.994,-46.993,-179.163,5.756,148.770
C03172=1199.913,59.245,-47.009,-179.161,5.757,148.769
C03173=1199.908,59.493,-47.026,-179.158,5.758,148.769
C03174=1199.903,59.743,-47.042,-179.155,5.758,148.768
C03175=1199.898,59.992,-47.059,-179.153,5.759,148.768
C03176=1199.893,60.241,-47.076,-179.150,5.760,148.767
C03177=1199.888,60.491,-47.092,-179.147,5.761,148.766
C03178=1199.883,60.740,-47.109,-179.145,5.762,148.766
C03179=1199.878,60.990,-47.125,-179.142,5.763,148.765
C03180=1199.873,61.240,-47.142,-179.140,5.763,148.765
C03181=1199.868,61.488,-47.158,-179.138,5.764,148.764
C03182=1199.864,61.738,-47.175,-179.134,5.765,148.763
C03183=1199.858,61.988,-47.192,-179.132,5.766,148.763
C03184=1199.853,62.236,-47.209,-179.130,5.767,148.762
C03185=1199.849,62.486,-47.225,-179.127,5.767,148.762
C03186=1199.844,62.736,-47.242,-179.124,5.768,148.761
C03187=1199.839,62.985,-47.259,-179.122,5.769,148.761
C03188=1199.834,63.234,-47.275,-179.119,5.770,148.760
C03189=1199.829,63.484,-47.293,-179.116,5.771,148.759
C03190=1199.824,63.733,-47.309,-179.114,5.772,148.759
C03191=1199.819,63.982,-47.326,-179.112,5.772,148.758
C03192=1199.814,64.232,-47.343,-179.109,5.773,148.758
C03193=1199.810,64.481,-47.360,-179.106,5.774,148.757
C03194=1199.804,64.730,-47.376,-179.104,5.775,148.756
C03195=1199.799,64.980,-47.393,-179.101,5.776,148.756
C03196=1199.795,65.229,-47.410,-179.099,5.776,148.755
C03197=1199.789,65.479,-47.427,-179.096,5.777,148.755
C03198=1199.785,65.728,-47.443,-179.093,5.778,148.754
C03199=1199.779,65.978,-47.461,-179.091,5.779,148.754
C03200=1199.775,66.227,-47.477,-179.088,5.780,148.753
C03201=1199.770,66.476,-47.494,-179.086,5.780,148.752
C03202=1199.765,66.726,-47.511,-179.084,5.781,148.752
C03203=1199.760,66.975,-47.528,-179.080,5.783,148.751
C03204=1199.755,67.225,-47.546,-179.078,5.783,148.751
C03205=1199.750,67.473,-47.562,-179.076,5.784,148.750
C03206=1199.745,67.723,-47.579,-179.073,5.785,148.749
C03207=1199.740,67.973,-47.596,-179.070,5.786,148.749
C03208=1199.735,68.222,-47.613,-179.068,5.787,148.748
C03209=1199.731,68.472,-47.630,-179.065,5.787,148.748
C03210=1199.725,68.720,-47.647,-179.063,5.788,148.747
C03211=1199.721,68.970,-47.664,-179.060,5.789,148.747
C03212=1199.716,69.220,-47.681,-179.057,5.790,148.746
C03213=1199.711,69.469,-47.698,-179.055,5.791,148.746
C03214=1199.705,69.718,-47.715,-179.052,5.792,148.745
C03215=1199.701,69.967,-47.732,-179.050,5.792,148.744
C03216=1199.696,70.217,-47.749,-179.047,5.794,148.744
C03217=1199.691,70.466,-47.766,-179.044,5.795,148.743
C03218=1199.686,70.716,-47.783,-179.042,5.795,148.742
C03219=1199.682,70.965,-47.801,-179.039,5.796,148.742
C03220=1199.676,71.214,-47.818,-179.037,5.797,148.741
C03221=1199.672,71.464,-47.834,-179.034,5.798,148.741
C03222=1199.666,71.713,-47.852,-179.031,5.799,148.740
C03223=1199.662,71.962,-47.869,-179.029,5.799,148.740
C03224=1199.657,72.212,-47.886,-179.027,5.800,148.739
C03225=1199.652,72.462,-47.904,-179.024,5.802,148.739
C03226=1199.647,72.710,-47.921,-179.021,5.802,148.738
C03227=1199.642,72.960,-47.938,-179.019,5.803,148.737
C03228=1199.637,73.209,-47.954,-179.016,5.804,148.737
C03229=1199.632,73.458,-47.972,-179.013,5.805,148.736
C03230=1199.627,73.708,-47.990,-179.011,5.806,148.736
C03231=1199.623,73.958,-48.006,-179.008,5.807,148.735
C03232=1199.617,74.206,-48.024,-179.006,5.807,148.735
C03233=1199.613,74.456,-48.041,-179.003,5.809,148.734
C03234=1199.608,74.705,-48.058,-179.000,5.809,148.733
C03235=1199.603,74.955,-48.076,-178.998,5.810,148.733
C03236=1199.598,75.204,-48.093,-178.995,5.811,148.732
C03237=1199.593,75.453,-48.111,-178.992,5.812,148.732
C03238=1199.588,75.703,-48.128,-178.990,5.813,148.731
C03239=1199.584,75.952,-48.145,-178.987,5.814,148.730
C03240=1199.579,76.202,-48.162,-178.985,5.815,148.730
C03241=1199.573,76.452,-48.180,-178.982,5.816,148.729
C03242=1199.569,76.700,-48.197,-178.979,5.817,148.729
C03243=1199.563,76.950,-48.214,-178.977,5.817,148.728
C03244=1199.558,77.199,-48.232,-178.975,5.818,148.728
C03245=1199.554,77.448,-48.249,-178.971,5.819,148.727
C03246=1199.549,77.697,-48.267,-178.969,5.820,148.727
C03247=1199.544,77.947,-48.284,-178.967,5.821,148.726
C03248=1199.539,78.196,-48.302,-178.964,5.823,148.725
C03249=1199.534,78.446,-48.319,-178.961,5.823,148.725
C03250=1199.530,78.695,-48.337,-178.959,5.824,148.724
C03251=1199.525,78.944,-48.355,-178.957,5.825,148.724
C03252=1199.519,79.194,-48.372,-178.953,5.826,148.723
C03253=1199.515,79.443,-48.389,-178.951,5.827,148.723
C03254=1199.510,79.693,-48.406,-178.949,5.827,148.722
C03255=1199.505,79.942,-48.424,-178.945,5.829,148.721
C03256=1199.500,80.192,-48.442,-178.943,5.830,148.721
C03257=1199.496,80.440,-48.459,-178.941,5.830,148.720
C03258=1199.490,80.709,-48.477,-178.937,5.832,148.720
C03259=1199.485,80.977,-48.497,-178.935,5.833,148.719
C03260=1199.480,81.245,-48.516,-178.933,5.833,148.719
C03261=1199.474,81.514,-48.535,-178.930,5.835,148.718
C03262=1199.469,81.763,-48.553,-178.927,5.835,148.717
C03263=1199.464,82.013,-48.570,-178.924,5.837,148.717
C03264=1199.460,82.262,-48.588,-178.922,5.837,148.716
C03265=1199.455,82.511,-48.606,-178.919,5.838,148.716
C03266=1199.450,82.761,-48.623,-178.917,5.839,148.715
C03267=1199.445,83.010,-48.641,-178.914,5.841,148.715
C03268=1199.440,83.259,-48.659,-178.911,5.841,148.714
C03269=1199.435,83.509,-48.676,-178.909,5.842,148.713
C03270=1199.430,83.758,-48.694,-178.906,5.843,148.713
C03271=1199.426,84.007,-48.711,-178.903,5.844,148.712
C03272=1199.421,84.256,-48.729,-178.901,5.845,148.712
C03273=1199.416,84.506,-48.747,-178.898,5.846,148.711
C03274=1199.411,84.755,-48.765,-178.896,5.847,148.711
C03275=1199.406,85.004,-48.783,-178.893,5.848,148.710
C03276=1199.401,85.254,-48.801,-178.890,5.849,148.709
C03277=1199.396,85.503,-48.819,-178.888,5.850,148.709
C03278=1199.391,85.752,-48.836,-178.885,5.851,148.708
C03279=1199.386,86.002,-48.854,-178.883,5.852,148.708
C03280=1199.381,86.251,-48.872,-178.880,5.853,148.707
C03281=1199.377,86.500,-48.889,-178.877,5.854,148.707
C03282=1199.372,86.750,-48.908,-178.875,5.854,148.706
C03283=1199.367,86.999,-48.925,-178.872,5.856,148.706
C03284=1199.362,87.249,-48.943,-178.870,5.857,148.705
C03285=1199.357,87.498,-48.961,-178.867,5.857,148.705
C03286=1199.352,87.747,-48.979,-178.865,5.859,148.704
C03287=1199.347,87.996,-48.997,-178.862,5.860,148.703
C03288=1199.343,88.245,-49.015,-178.859,5.860,148.703
C03289=1199.338,88.494,-49.033,-178.857,5.862,148.702
C03290=1199.333,88.744,-49.051,-178.854,5.863,148.702
C03291=1199.328,88.993,-49.069,-178.852,5.863,148.701
C03292=1199.323,89.243,-49.086,-178.849,5.865,148.701
C03293=1199.318,89.492,-49.104,-178.847,5.866,148.700
C03294=1199.313,89.742,-49.122,-178.844,5.866,148.700
C03295=1199.308,89.991,-49.140,-178.841,5.868,148.699
C03296=1199.304,90.240,-49.158,-178.839,5.869,148.699
C03297=1199.299,90.489,-49.176,-178.836,5.869,148.698
C03298=1199.294,90.738,-49.194,-178.833,5.871,148.697
C03299=1199.289,90.987,-49.212,-178.831,5.872,148.697
C03300=1199.284,91.238,-49.231,-178.828,5.873,148.696
C03301=1199.279,91.487,-49.249,-178.825,5.874,148.696
C03302=1199.274,91.736,-49.267,-178.823,5.875,148.695
C03303=1199.269,91.985,-49.285,-178.820,5.876,148.695
C03304=1199.264,92.234,-49.303,-178.818,5.877,148.694
C03305=1199.259,92.484,-49.321,-178.815,5.878,148.694
C03306=1199.255,92.733,-49.339,-178.813,5.879,148.693
C03307=1199.250,92.982,-49.358,-178.810,5.880,148.693
C03308=1199.245,93.231,-49.376,-178.807,5.880,148.692
C03309=1199.240,93.480,-49.394,-178.805,5.882,148.692
C03310=1199.236,93.730,-49.412,-178.802,5.883,148.691
C03311=1199.231,93.980,-49.431,-178.800,5.884,148.690
C03312=1199.226,94.229,-49.449,-178.797,5.885,148.690
C03313=1199.221,94.478,-49.467,-178.795,5.886,148.689
C03314=1199.216,94.727,-49.485,-178.791,5.887,148.689
C03315=1199.211,94.976,-49.503,-178.789,5.888,148.688
C03316=1199.207,95.226,-49.522,-178.787,5.889,148.688
C03317=1199.201,95.475,-49.540,-178.784,5.891,148.687
C03318=1199.196,95.724,-49.558,-178.781,5.891,148.687
C03319=1199.191,95.974,-49.576,-178.779,5.892,148.686
C03320=1199.187,96.223,-49.595,-178.776,5.894,148.686
C03321=1199.182,96.473,-49.613,-178.774,5.894,148.685
C03322=1199.178,96.721,-49.631,-178.771,5.896,148.684
C03323=1199.172,96.971,-49.650,-178.769,5.897,148.684
C03324=1199.168,97.220,-49.668,-178.766,5.897,148.683
C03325=1199.163,97.470,-49.686,-178.763,5.899,148.683
C03326=1199.158,97.718,-49.705,-178.761,5.900,148.682
C03327=1199.152,97.968,-49.724,-178.757,5.901,148.682
C03328=1199.148,98.218,-49.742,-178.755,5.902,148.681
C03329=1199.143,98.467,-49.760,-178.753,5.903,148.681
C03330=1199.139,98.715,-49.779,-178.750,5.904,148.680
C03331=1199.133,98.965,-49.797,-178.747,5.905,148.680
C03332=1199.129,99.215,-49.816,-178.745,5.907,148.679
C03333=1199.124,99.463,-49.834,-178.742,5.907,148.679
C03334=1199.119,99.712,-49.852,-178.740,5.908,148.678
C03335=1199.114,99.963,-49.871,-178.737,5.910,148.677
C03336=1199.109,100.211,-49.890,-178.735,5.910,148.677
C03337=1199.105,100.460,-49.908,-178.731,5.912,148.676
C03338=1199.099,100.710,-49.926,-178.729,5.913,148.676
C03339=1199.095,100.959,-49.945,-178.727,5.913,148.675
C03340=1199.090,101.208,-49.963,-178.724,5.915,148.675
C03341=1199.084,101.458,-49.982,-178.721,5.916,148.674
C03342=1199.080,101.707,-50.001,-178.719,5.917,148.674
C03343=1199.075,101.956,-50.019,-178.716,5.918,148.673
C03344=1199.070,102.205,-50.038,-178.714,5.919,148.673
C03345=1199.066,102.455,-50.057,-178.711,5.920,148.672
C03346=1199.061,102.703,-50.075,-178.709,5.921,148.672
C03347=1199.056,102.953,-50.094,-178.705,5.923,148.671
C03348=1199.051,103.203,-50.112,-178.703,5.924,148.671
C03349=1199.047,103.451,-50.131,-178.701,5.924,148.670
C03350=1199.042,103.702,-50.150,-178.698,5.926,148.670
C03351=1199.037,103.950,-50.169,-178.695,5.927,148.669
C03352=1199.031,104.200,-50.187,-178.693,5.928,148.669
C03353=1199.027,104.449,-50.206,-178.690,5.929,148.668
C03354=1199.022,104.698,-50.224,-178.687,5.931,148.668
C03355=1199.017,104.947,-50.244,-178.685,5.931,148.667
C03356=1199.013,105.197,-50.262,-178.682,5.933,148.667
C03357=1199.007,105.446,-50.281,-178.680,5.934,148.666
C03358=1199.003,105.695,-50.300,-178.677,5.934,148.665
C03359=1198.998,105.944,-50.319,-178.674,5.936,148.665
C03360=1198.993,106.193,-50.337,-178.672,5.937,148.664
C03361=1198.988,106.443,-50.356,-178.669,5.939,148.664
C03362=1198.983,106.711,-50.377,-178.667,5.939,148.663
C03363=1198.978,106.980,-50.397,-178.663,5.941,148.663
C03364=1198.973,107.248,-50.417,-178.661,5.942,148.662
C03365=1198.967,107.516,-50.437,-178.658,5.943,148.662
C03366=1198.963,107.766,-50.457,-178.655,5.945,148.661
C03367=1198.958,108.014,-50.475,-178.653,5.945,148.661
C03368=1198.953,108.265,-50.494,-178.650,5.947,148.660
C03369=1198.948,108.513,-50.513,-178.647,5.948,148.660
C03370=1198.943,108.762,-50.532,-178.645,5.949,148.659
C03371=1198.939,109.012,-50.551,-178.642,5.950,148.659
C03372=1198.933,109.261,-50.570,-178.640,5.951,148.658
C03373=1198.929,109.510,-50.589,-178.637,5.952,148.658
C03374=1198.924,109.759,-50.608,-178.635,5.953,148.657
C03375=1198.920,110.009,-50.627,-178.631,5.955,148.656
C03376=1198.914,110.258,-50.646,-178.629,5.955,148.656
C03377=1198.910,110.507,-50.666,-178.626,5.957,148.655
C03378=1198.905,110.756,-50.684,-178.624,5.958,148.655
C03379=1198.900,111.006,-50.703,-178.621,5.960,148.655
C03380=1198.895,111.254,-50.722,-178.619,5.960,148.654
C03381=1198.891,111.504,-50.742,-178.616,5.962,148.654
C03382=1198.886,111.753,-50.760,-178.613,5.963,148.653
C03383=1198.881,112.003,-50.779,-178.611,5.964,148.653
C03384=1198.876,112.252,-50.799,-178.608,5.965,148.652
C03385=1198.872,112.501,-50.818,-178.605,5.967,148.651
C03386=1198.866,112.750,-50.837,-178.603,5.967,148.651
C03387=1198.861,113.000,-50.856,-178.601,5.968,148.650
C03388=1198.857,113.249,-50.875,-178.598,5.970,148.650
C03389=1198.852,113.498,-50.894,-178.595,5.970,148.649
C03390=1198.847,113.747,-50.913,-178.593,5.972,148.649
C03391=1198.843,113.996,-50.933,-178.590,5.973,148.648
C03392=1198.837,114.245,-50.952,-178.587,5.975,148.648
C03393=1198.833,114.495,-50.971,-178.585,5.975,148.647
C03394=1198.828,114.743,-50.990,-178.582,5.977,148.647
C03395=1198.823,114.993,-51.009,-178.580,5.978,148.647
C03396=1198.818,115.243,-51.029,-178.577,5.979,148.646
C03397=1198.814,115.492,-51.047,-178.575,5.980,148.645
C03398=1198.809,115.741,-51.067,-178.571,5.982,148.645
C03399=1198.803,115.990,-51.086,-178.569,5.983,148.644
C03400=1198.799,116.239,-51.105,-178.566,5.984,148.644
C03401=1198.794,116.488,-51.125,-178.564,5.985,148.643
C03402=1198.789,116.738,-51.144,-178.561,5.987,148.643
C03403=1198.785,116.987,-51.164,-178.559,5.987,148.642
C03404=1198.780,117.236,-51.183,-178.556,5.989,148.642
C03405=1198.775,117.485,-51.202,-178.553,5.990,148.641
C03406=1198.770,117.734,-51.222,-178.551,5.991,148.641
C03407=1198.765,117.984,-51.241,-178.549,5.992,148.641
C03408=1198.760,118.233,-51.261,-178.545,5.994,148.640
C03409=1198.756,118.482,-51.280,-178.543,5.995,148.639
C03410=1198.751,118.731,-51.299,-178.540,5.996,148.639
C03411=1198.746,118.980,-51.319,-178.537,5.998,148.638
C03412=1198.741,119.229,-51.339,-178.535,5.999,148.638
C03413=1198.737,119.479,-51.359,-178.532,6.000,148.637
C03414=1198.732,119.727,-51.377,-178.530,6.001,148.637
C03415=1198.727,119.977,-51.397,-178.527,6.003,148.636
C03416=1198.722,120.227,-51.417,-178.525,6.003,148.636
C03417=1198.717,120.475,-51.436,-178.522,6.005,148.636
C03418=1198.712,120.725,-51.456,-178.519,6.006,148.635
C03419=1198.708,120.975,-51.475,-178.517,6.008,148.635
C03420=1198.703,121.222,-51.495,-178.514,6.008,148.634
C03421=1198.699,121.472,-51.514,-178.511,6.010,148.634
C03422=1198.694,121.722,-51.534,-178.509,6.011,148.633
C03423=1198.689,121.970,-51.553,-178.506,6.012,148.632
C03424=1198.684,122.220,-51.573,-178.504,6.013,148.632
C03425=1198.679,122.470,-51.593,-178.501,6.015,148.631
C03426=1198.674,122.718,-51.613,-178.498,6.016,148.631
C03427=1198.669,122.967,-51.632,-178.496,6.017,148.631
C03428=1198.665,123.217,-51.651,-178.493,6.019,148.630
C03429=1198.660,123.466,-51.671,-178.491,6.020,148.630
C03430=1198.655,123.715,-51.691,-178.487,6.021,148.629
C03431=1198.651,123.964,-51.711,-178.485,6.022,148.629
C03432=1198.646,124.214,-51.730,-178.483,6.024,148.628
C03433=1198.641,124.463,-51.750,-178.480,6.024,148.628
C03434=1198.636,124.711,-51.770,-178.477,6.026,148.627
C03435=1198.631,124.961,-51.790,-178.475,6.027,148.627
C03436=1198.626,125.210,-51.809,-178.472,6.029,148.626
C03437=1198.622,125.459,-51.829,-178.469,6.030,148.626
C03438=1198.617,125.708,-51.849,-178.467,6.031,148.625
C03439=1198.612,125.958,-51.869,-178.464,6.033,148.625
C03440=1198.607,126.206,-51.889,-178.462,6.034,148.624
C03441=1198.602,126.456,-51.908,-178.459,6.035,148.624
C03442=1198.598,126.705,-51.929,-178.457,6.036,148.623
C03443=1198.593,126.954,-51.948,-178.454,6.038,148.623
C03444=1198.588,127.204,-51.968,-178.451,6.039,148.622
C03445=1198.583,127.452,-51.988,-178.449,6.040,148.622
C03446=1198.579,127.702,-52.008,-178.446,6.042,148.621
C03447=1198.574,127.951,-52.028,-178.443,6.042,148.621
C03448=1198.570,128.200,-52.048,-178.441,6.044,148.620
C03449=1198.564,128.449,-52.067,-178.439,6.045,148.620
C03450=1198.560,128.698,-52.087,-178.435,6.047,148.619
C03451=1198.555,128.948,-52.107,-178.433,6.048,148.619
C03452=1198.551,129.197,-52.127,-178.431,6.049,148.619
C03453=1198.546,129.446,-52.147,-178.427,6.051,148.618
C03454=1198.541,129.694,-52.167,-178.425,6.052,148.618
C03455=1198.536,129.944,-52.187,-178.422,6.053,148.617
C03456=1198.531,130.193,-52.208,-178.419,6.055,148.617
C03457=1198.526,130.443,-52.227,-178.417,6.056,148.616
C03458=1198.522,130.692,-52.248,-178.414,6.057,148.616
C03459=1198.517,130.941,-52.267,-178.412,6.058,148.615
C03460=1198.512,131.190,-52.287,-178.409,6.060,148.615
C03461=1198.507,131.438,-52.308,-178.406,6.061,148.614
C03462=1198.503,131.688,-52.327,-178.404,6.062,148.614
C03463=1198.498,131.937,-52.348,-178.401,6.064,148.613
C03464=1198.493,132.187,-52.368,-178.399,6.065,148.613
C03465=1198.488,132.436,-52.388,-178.396,6.066,148.612
C03466=1198.483,132.704,-52.409,-178.393,6.068,148.612
C03467=1198.478,132.973,-52.432,-178.390,6.070,148.611
C03468=1198.473,133.241,-52.453,-178.388,6.071,148.611
C03469=1198.468,133.510,-52.475,-178.385,6.072,148.610
C03470=1198.463,133.759,-52.495,-178.382,6.074,148.610
C03471=1198.459,134.008,-52.515,-178.380,6.074,148.609
C03472=1198.453,134.258,-52.536,-178.377,6.076,148.609
C03473=1198.448,134.506,-52.556,-178.374,6.078,148.609
C03474=1198.444,134.755,-52.576,-178.372,6.079,148.608
C03475=1198.439,135.004,-52.596,-178.369,6.080,148.608
C03476=1198.434,135.254,-52.617,-178.366,6.082,148.607
C03477=1198.429,135.503,-52.637,-178.364,6.083,148.607
C03478=1198.425,135.752,-52.657,-178.361,6.084,148.606
C03479=1198.420,136.001,-52.678,-178.359,6.085,148.606
C03480=1198.415,136.251,-52.698,-178.356,6.087,148.605
C03481=1198.411,136.500,-52.718,-178.353,6.089,148.605
C03482=1198.406,136.749,-52.739,-178.351,6.090,148.604
C03483=1198.402,136.998,-52.759,-178.348,6.091,148.604
C03484=1198.397,137.247,-52.780,-178.345,6.093,148.603
C03485=1198.392,137.497,-52.800,-178.343,6.094,148.603
C03486=1198.387,137.745,-52.820,-178.340,6.096,148.603
C03487=1198.382,137.994,-52.841,-178.338,6.096,148.602
C03488=1198.377,138.243,-52.861,-178.335,6.098,148.602
C03489=1198.373,138.492,-52.881,-178.332,6.100,148.601
C03490=1198.367,138.741,-52.902,-178.330,6.101,148.601
C03491=1198.363,138.990,-52.923,-178.327,6.102,148.600
C03492=1198.358,139.240,-52.942,-178.324,6.104,148.600
C03493=1198.353,139.489,-52.963,-178.322,6.105,148.599
C03494=1198.349,139.738,-52.984,-178.319,6.107,148.599
C03495=1198.344,139.987,-53.004,-178.316,6.108,148.598
C03496=1198.339,140.236,-53.025,-178.314,6.109,148.598
C03497=1198.335,140.485,-53.045,-178.311,6.111,148.598
C03498=1198.329,140.734,-53.066,-178.308,6.112,148.597
C03499=1198.325,140.983,-53.087,-178.306,6.113,148.597
C03500=1198.321,141.232,-53.107,-178.303,6.115,148.596
C03501=1198.315,141.482,-53.128,-178.301,6.117,148.596
C03502=1198.311,141.731,-53.149,-178.298,6.117,148.595
C03503=1198.306,141.980,-53.169,-178.296,6.119,148.595
C03504=1198.301,142.229,-53.190,-178.293,6.121,148.594
C03505=1198.297,142.478,-53.210,-178.291,6.122,148.594
C03506=1198.292,142.727,-53.231,-178.288,6.123,148.593
C03507=1198.288,142.977,-53.252,-178.285,6.125,148.593
C03508=1198.283,143.226,-53.273,-178.283,6.126,148.593
C03509=1198.278,143.475,-53.293,-178.280,6.127,148.592
C03510=1198.273,143.724,-53.314,-178.277,6.129,148.592
C03511=1198.269,143.973,-53.335,-178.275,6.130,148.591
C03512=1198.264,144.222,-53.356,-178.272,6.132,148.591
C03513=1198.259,144.471,-53.376,-178.269,6.133,148.590
C03514=1198.254,144.720,-53.397,-178.267,6.134,148.590
C03515=1198.250,144.969,-53.418,-178.264,6.136,148.589
C03516=1198.245,145.218,-53.439,-178.261,6.138,148.589
C03517=1198.240,145.467,-53.459,-178.259,6.138,148.588
C03518=1198.235,145.716,-53.480,-178.256,6.140,148.588
C03519=1198.231,145.965,-53.501,-178.254,6.142,148.588
C03520=1198.226,146.215,-53.522,-178.251,6.144,148.587
C03521=1198.222,146.464,-53.542,-178.248,6.144,148.587
C03522=1198.217,146.713,-53.564,-178.246,6.146,148.586
C03523=1198.212,146.962,-53.585,-178.243,6.148,148.586
C03524=1198.207,147.211,-53.605,-178.241,6.149,148.586
C03525=1198.202,147.460,-53.626,-178.238,6.150,148.585
C03526=1198.198,147.709,-53.647,-178.235,6.152,148.585
C03527=1198.193,147.958,-53.668,-178.233,6.153,148.584
C03528=1198.188,148.207,-53.689,-178.230,6.155,148.584
C03529=1198.184,148.457,-53.710,-178.227,6.157,148.583
C03530=1198.179,148.705,-53.732,-178.224,6.158,148.583
C03531=1198.174,148.954,-53.752,-178.222,6.159,148.582
C03532=1198.169,149.204,-53.773,-178.219,6.161,148.582
C03533=1198.164,149.453,-53.794,-178.217,6.163,148.582
C03534=1198.160,149.701,-53.815,-178.214,6.163,148.581
C03535=1198.155,149.951,-53.837,-178.212,6.165,148.581
C03536=1198.150,150.200,-53.857,-178.209,6.167,148.580
C03537=1198.146,150.449,-53.879,-178.206,6.169,148.580
C03538=1198.141,150.698,-53.900,-178.204,6.170,148.580
C03539=1198.136,150.947,-53.921,-178.201,6.171,148.579
C03540=1198.131,151.196,-53.942,-178.198,6.173,148.579
C03541=1198.127,151.446,-53.963,-178.196,6.174,148.578
C03542=1198.122,151.694,-53.985,-178.193,6.175,148.578
C03543=1198.118,151.943,-54.005,-178.190,6.177,148.577
C03544=1198.112,152.192,-54.026,-178.188,6.179,148.577
C03545=1198.108,152.441,-54.048,-178.185,6.180,148.576
C03546=1198.103,152.691,-54.069,-178.183,6.181,148.576
C03547=1198.099,152.939,-54.090,-178.180,6.183,148.576
C03548=1198.094,153.189,-54.111,-178.177,6.185,148.575
C03549=1198.089,153.437,-54.133,-178.175,6.186,148.575
C03550=1198.084,153.687,-54.154,-178.172,6.187,148.574
C03551=1198.080,153.936,-54.175,-178.169,6.189,148.574
C03552=1198.075,154.185,-54.196,-178.167,6.191,148.574
C03553=1198.070,154.433,-54.218,-178.164,6.192,148.573
C03554=1198.065,154.683,-54.239,-178.162,6.193,148.573
C03555=1198.061,154.932,-54.260,-178.159,6.195,148.572
C03556=1198.056,155.181,-54.281,-178.156,6.197,148.572
C03557=1198.051,155.430,-54.303,-178.154,6.198,148.571
C03558=1198.047,155.680,-54.324,-178.151,6.200,148.571
C03559=1198.042,155.928,-54.346,-178.148,6.201,148.570
C03560=1198.037,156.177,-54.367,-178.146,6.203,148.570
C03561=1198.033,156.426,-54.388,-178.143,6.204,148.570
C03562=1198.028,156.675,-54.410,-178.141,6.206,148.569
C03563=1198.023,156.924,-54.431,-178.138,6.207,148.569
C03564=1198.018,157.173,-54.453,-178.135,6.209,148.568
C03565=1198.014,157.422,-54.475,-178.133,6.210,148.568
C03566=1198.009,157.672,-54.496,-178.130,6.212,148.568
C03567=1198.004,157.920,-54.517,-178.127,6.213,148.567
C03568=1198.000,158.169,-54.539,-178.125,6.215,148.567
C03569=1197.995,158.419,-54.560,-178.122,6.217,148.566
C03570=1197.990,158.688,-54.583,-178.119,6.218,148.566
C03571=1197.985,158.956,-54.607,-178.116,6.220,148.565
C03572=1197.980,159.226,-54.630,-178.114,6.222,148.565
C03573=1197.975,159.495,-54.653,-178.110,6.223,148.564
C03574=1197.970,159.743,-54.674,-178.108,6.224,148.564
C03575=1197.965,159.992,-54.696,-178.106,6.226,148.564
C03576=1197.961,160.241,-54.718,-178.103,6.228,148.563
C03577=1197.956,160.491,-54.739,-178.100,6.230,148.563
C03578=1197.951,160.739,-54.761,-178.097,6.231,148.562
C03579=1197.947,160.989,-54.783,-178.095,6.232,148.562
C03580=1197.942,161.237,-54.804,-178.092,6.234,148.562
C03581=1197.938,161.487,-54.827,-178.090,6.236,148.561
C03582=1197.932,161.736,-54.848,-178.087,6.238,148.561
C03583=1197.928,161.985,-54.869,-178.085,6.239,148.560
C03584=1197.923,162.234,-54.891,-178.082,6.240,148.560
C03585=1197.918,162.482,-54.913,-178.079,6.242,148.560
C03586=1197.914,162.732,-54.935,-178.076,6.244,148.559
C03587=1197.909,162.980,-54.957,-178.074,6.245,148.559
C03588=1197.904,163.230,-54.978,-178.072,6.246,148.558
C03589=1197.900,163.479,-55.000,-178.069,6.248,148.558
C03590=1197.895,163.728,-55.021,-178.066,6.250,148.558
C03591=1197.891,163.977,-55.043,-178.064,6.252,148.557
C03592=1197.886,164.226,-55.065,-178.061,6.254,148.557
C03593=1197.881,164.474,-55.087,-178.058,6.255,148.556
C03594=1197.877,164.724,-55.109,-178.056,6.256,148.556
C03595=1197.872,164.972,-55.130,-178.053,6.258,148.556
C03596=1197.868,165.222,-55.153,-178.050,6.260,148.555
C03597=1197.862,165.471,-55.175,-178.048,6.261,148.555
C03598=1197.858,165.720,-55.197,-178.045,6.263,148.554
C03599=1197.853,165.969,-55.219,-178.043,6.264,148.554
C03600=1197.849,166.218,-55.241,-178.040,6.266,148.554
C03601=1197.844,166.467,-55.262,-178.037,6.267,148.553
C03602=1197.839,166.716,-55.284,-178.034,6.269,148.553
C03603=1197.835,166.965,-55.306,-178.032,6.271,148.552
C03604=1197.830,167.214,-55.328,-178.029,6.273,148.552
C03605=1197.825,167.463,-55.350,-178.027,6.274,148.552
C03606=1197.820,167.711,-55.372,-178.024,6.275,148.551
C03607=1197.816,167.961,-55.394,-178.022,6.277,148.551
C03608=1197.811,168.209,-55.416,-178.019,6.279,148.551
C03609=1197.806,168.459,-55.438,-178.016,6.281,148.550
C03610=1197.802,168.707,-55.460,-178.013,6.282,148.550
C03611=1197.797,168.956,-55.483,-178.010,6.284,148.549
C03612=1197.792,169.205,-55.505,-178.008,6.285,148.549
C03613=1197.788,169.454,-55.527,-178.006,6.287,148.548
C03614=1197.783,169.704,-55.549,-178.003,6.289,148.548
C03615=1197.779,169.952,-55.570,-178.000,6.290,148.548
C03616=1197.774,170.202,-55.593,-177.998,6.292,148.547
C03617=1197.769,170.450,-55.615,-177.995,6.294,148.547
C03618=1197.765,170.699,-55.637,-177.993,6.295,148.547
C03619=1197.760,170.948,-55.659,-177.990,6.297,148.546
C03620=1197.755,171.198,-55.682,-177.988,6.299,148.546
C03621=1197.750,171.446,-55.703,-177.984,6.300,148.545
C03622=1197.746,171.695,-55.726,-177.982,6.302,148.545
C03623=1197.741,171.944,-55.748,-177.979,6.304,148.545
C03624=1197.736,172.193,-55.770,-177.976,6.305,148.544
C03625=1197.732,172.442,-55.793,-177.974,6.307,148.544
C03626=1197.727,172.691,-55.815,-177.972,6.308,148.543
C03627=1197.722,172.940,-55.838,-177.969,6.310,148.543
C03628=1197.717,173.189,-55.859,-177.966,6.312,148.543
C03629=1197.713,173.438,-55.882,-177.964,6.314,148.542
C03630=1197.708,173.687,-55.904,-177.961,6.315,148.542
C03631=1197.704,173.936,-55.926,-177.958,6.317,148.542
C03632=1197.700,174.185,-55.949,-177.956,6.319,148.541
C03633=1197.694,174.434,-55.971,-177.953,6.321,148.541
C03634=1197.690,174.683,-55.993,-177.951,6.322,148.541
C03635=1197.686,174.932,-56.016,-177.948,6.323,148.540
C03636=1197.680,175.181,-56.038,-177.945,6.325,148.540
C03637=1197.676,175.429,-56.061,-177.942,6.327,148.539
C03638=1197.671,175.678,-56.084,-177.940,6.329,148.539
C03639=1197.666,175.928,-56.106,-177.937,6.330,148.539
C03640=1197.662,176.176,-56.128,-177.934,6.332,148.538
C03641=1197.657,176.425,-56.151,-177.932,6.334,148.538
C03642=1197.653,176.674,-56.173,-177.929,6.336,148.537
C03643=1197.648,176.924,-56.196,-177.927,6.337,148.537
C03644=1197.643,177.172,-56.218,-177.924,6.339,148.537
C03645=1197.639,177.421,-56.240,-177.922,6.340,148.536
C03646=1197.634,177.670,-56.264,-177.919,6.342,148.536
C03647=1197.629,177.919,-56.285,-177.916,6.344,148.536
C03648=1197.625,178.168,-56.309,-177.914,6.346,148.535
C03649=1197.620,178.417,-56.331,-177.911,6.348,148.535
C03650=1197.615,178.666,-56.354,-177.908,6.349,148.535
C03651=1197.611,178.915,-56.376,-177.906,6.351,148.534
C03652=1197.606,179.164,-56.399,-177.903,6.353,148.534
C03653=1197.602,179.412,-56.422,-177.901,6.354,148.533
C03654=1197.597,179.662,-56.444,-177.898,6.356,148.533
C03655=1197.593,179.910,-56.467,-177.896,6.358,148.533
